C01819=1209.672,408.149,-82.083,-175.808,8.325,148.423
C01820=1209.667,408.397,-82.117,-175.807,8.328,148.423
C01821=1209.664,408.644,-82.152,-175.807,8.330,148.424
C01822=1209.660,408.891,-82.187,-175.807,8.333,148.424
C01823=1209.656,409.139,-82.222,-175.806,8.335,148.425
C01824=1209.651,409.386,-82.257,-175.806,8.337,148.425
C01825=1209.647,409.634,-82.291,-175.806,8.339,148.426
C01826=1209.644,409.882,-82.327,-175.805,8.341,148.426
C01827=1209.639,410.129,-82.361,-175.805,8.343,148.427
C01828=1209.636,410.377,-82.397,-175.804,8.346,148.427
C01829=1209.631,410.624,-82.431,-175.804,8.348,148.428
C01830=1209.627,410.871,-82.467,-175.804,8.350,148.428
C01831=1209.623,411.120,-82.502,-175.803,8.352,148.429
C01832=1209.619,411.366,-82.537,-175.802,8.355,148.429
C01833=1209.615,411.615,-82.572,-175.802,8.357,148.430
C01834=1209.612,411.861,-82.606,-175.802,8.359,148.430
C01835=1209.608,412.109,-82.642,-175.801,8.361,148.430
C01836=1209.604,412.357,-82.677,-175.801,8.364,148.431
C01837=1209.600,412.603,-82.712,-175.801,8.366,148.431
C01838=1209.596,412.852,-82.747,-175.800,8.368,148.432
C01839=1209.592,413.098,-82.782,-175.800,8.370,148.432
C01840=1209.588,413.346,-82.817,-175.800,8.372,148.433
C01841=1209.584,413.594,-82.852,-175.799,8.374,148.433
C01842=1209.579,413.841,-82.887,-175.799,8.377,148.434
C01843=1209.576,414.089,-82.922,-175.798,8.379,148.434
C01844=1209.571,414.336,-82.957,-175.798,8.381,148.435
C01845=1209.567,414.584,-82.992,-175.798,8.383,148.435
C01846=1209.564,414.831,-83.028,-175.797,8.385,148.435
C01847=1209.559,415.079,-83.062,-175.797,8.387,148.436
C01848=1209.556,415.326,-83.098,-175.796,8.390,148.437
C01849=1209.552,415.574,-83.133,-175.796,8.392,148.437
C01850=1209.547,415.821,-83.168,-175.796,8.394,148.437
C01851=1209.544,416.069,-83.204,-175.795,8.396,148.438
C01852=1209.539,416.325,-83.240,-175.795,8.398,148.438
C01853=1209.535,416.581,-83.276,-175.795,8.400,148.439
C01854=1209.533,416.838,-83.312,-175.794,8.402,148.439
C01855=1209.535,417.093,-83.348,-175.794,8.404,148.440
C01856=1209.114,417.093,-83.384,-175.797,8.414,148.443
C01857=1209.112,416.835,-83.348,-175.797,8.413,148.443
C01858=1209.113,416.576,-83.312,-175.798,8.411,148.442
C01859=1209.118,416.317,-83.275,-175.798,8.409,148.442
C01860=1209.122,416.058,-83.238,-175.798,8.407,148.441
C01861=1209.126,415.811,-83.203,-175.799,8.405,148.441
C01862=1209.130,415.563,-83.168,-175.799,8.402,148.441
C01863=1209.134,415.315,-83.133,-175.799,8.400,148.440
C01864=1209.138,415.068,-83.097,-175.800,8.398,148.440
C01865=1209.142,414.820,-83.063,-175.800,8.396,148.439
C01866=1209.146,414.573,-83.027,-175.801,8.394,148.439
C01867=1209.150,414.325,-82.993,-175.801,8.392,148.438
C01868=1209.154,414.078,-82.957,-175.801,8.389,148.438
C01869=1209.158,413.831,-82.922,-175.802,8.387,148.437
C01870=1209.162,413.583,-82.887,-175.802,8.385,148.437
C01871=1209.166,413.335,-82.851,-175.802,8.383,148.436
C01872=1209.170,413.088,-82.817,-175.803,8.381,148.436
C01873=1209.173,412.841,-82.782,-175.803,8.379,148.435
C01874=1209.178,412.593,-82.748,-175.803,8.376,148.435
C01875=1209.181,412.346,-82.712,-175.804,8.374,148.435
C01876=1209.185,412.098,-82.677,-175.804,8.372,148.434
C01877=1209.190,411.851,-82.642,-175.805,8.370,148.434
C01878=1209.193,411.603,-82.607,-175.805,8.368,148.433
C01879=1209.198,411.356,-82.572,-175.805,8.366,148.433
C01880=1209.201,411.108,-82.536,-175.806,8.363,148.432
C01881=1209.205,410.860,-82.502,-175.807,8.360,148.432
C01882=1209.210,410.614,-82.466,-175.807,8.358,148.431
C01883=1209.214,410.365,-82.432,-175.807,8.356,148.431
C01884=1209.218,410.119,-82.396,-175.808,8.354,148.430
C01885=1209.222,409.871,-82.362,-175.808,8.352,148.430
C01886=1209.226,409.623,-82.326,-175.808,8.349,148.429
C01887=1209.230,409.376,-82.292,-175.809,8.347,148.429
C01888=1209.234,409.128,-82.256,-175.809,8.345,148.428
C01889=1209.238,408.881,-82.222,-175.810,8.343,148.428
C01890=1209.242,408.633,-82.186,-175.810,8.341,148.428
C01891=1209.246,408.386,-82.152,-175.810,8.339,148.427
C01892=1209.250,408.138,-82.117,-175.811,8.336,148.426
C01893=1209.253,407.890,-82.082,-175.812,8.334,148.426
C01894=1209.258,407.643,-82.047,-175.812,8.331,148.426
C01895=1209.262,407.396,-82.012,-175.812,8.329,148.425
C01896=1209.266,407.148,-81.977,-175.813,8.327,148.425
C01897=1209.270,406.901,-81.942,-175.813,8.325,148.424
C01898=1209.275,406.653,-81.907,-175.813,8.323,148.424
C01899=1209.278,406.405,-81.872,-175.814,8.320,148.423
C01900=1209.281,406.158,-81.838,-175.814,8.318,148.423
C01901=1209.286,405.910,-81.803,-175.815,8.315,148.422
C01902=1209.290,405.663,-81.768,-175.815,8.313,148.422
C01903=1209.294,405.416,-81.733,-175.816,8.311,148.421
C01904=1209.298,405.167,-81.698,-175.816,8.309,148.421
C01905=1209.302,404.921,-81.663,-175.816,8.306,148.420
C01906=1209.306,404.672,-81.628,-175.817,8.304,148.420
C01907=1209.311,404.426,-81.593,-175.818,8.301,148.419
C01908=1209.314,404.178,-81.559,-175.818,8.299,148.419
C01909=1209.318,403.930,-81.524,-175.819,8.297,148.418
C01910=1209.322,403.683,-81.489,-175.819,8.295,148.418
C01911=1209.326,403.435,-81.454,-175.820,8.292,148.417
C01912=1209.331,403.187,-81.419,-175.820,8.289,148.417
C01913=1209.334,402.940,-81.384,-175.820,8.287,148.416
C01914=1209.338,402.693,-81.350,-175.821,8.285,148.416
C01915=1209.342,402.445,-81.315,-175.821,8.282,148.415
C01916=1209.346,402.198,-81.280,-175.822,8.280,148.415
C01917=1209.350,401.950,-81.245,-175.822,8.278,148.414
C01918=1209.355,401.702,-81.211,-175.822,8.276,148.414
C01919=1209.359,401.455,-81.175,-175.824,8.273,148.414
C01920=1209.362,401.208,-81.141,-175.824,8.271,148.413
C01921=1209.366,400.960,-81.106,-175.824,8.268,148.412
C01922=1209.371,400.712,-81.072,-175.825,8.266,148.412
C01923=1209.375,400.465,-81.036,-175.825,8.263,148.412
C01924=1209.379,400.217,-81.002,-175.826,8.261,148.411
C01925=1209.382,399.969,-80.968,-175.826,8.259,148.411
C01926=1209.387,399.722,-80.933,-175.827,8.256,148.410
C01927=1209.391,399.475,-80.898,-175.827,8.254,148.410
C01928=1209.395,399.227,-80.863,-175.828,8.251,148.409
C01929=1209.399,398.979,-80.828,-175.829,8.248,148.409
C01930=1209.403,398.732,-80.795,-175.829,8.246,148.408
C01931=1209.407,398.484,-80.759,-175.829,8.244,148.408
C01932=1209.411,398.237,-80.725,-175.830,8.241,148.407
C01933=1209.415,397.989,-80.690,-175.831,8.239,148.407
C01934=1209.419,397.742,-80.656,-175.831,8.236,148.406
C01935=1209.423,397.494,-80.620,-175.832,8.234,148.406
C01936=1209.427,397.247,-80.586,-175.832,8.232,148.405
C01937=1209.431,396.999,-80.551,-175.833,8.228,148.405
C01938=1209.435,396.752,-80.517,-175.834,8.226,148.404
C01939=1209.439,396.503,-80.482,-175.834,8.223,148.404
C01940=1209.444,396.256,-80.448,-175.835,8.221,148.403
C01941=1209.447,396.009,-80.412,-175.836,8.218,148.403
C01942=1209.451,395.761,-80.378,-175.836,8.216,148.402
C01943=1209.456,395.514,-80.344,-175.836,8.214,148.402
C01944=1209.460,395.266,-80.309,-175.837,8.211,148.401
C01945=1209.464,395.018,-80.275,-175.838,8.209,148.401
C01946=1209.467,394.771,-80.240,-175.839,8.206,148.400
C01947=1209.472,394.523,-80.206,-175.839,8.204,148.400
C01948=1209.476,394.276,-80.170,-175.840,8.200,148.399
C01949=1209.480,394.029,-80.137,-175.840,8.198,148.399
C01950=1209.484,393.781,-80.102,-175.841,8.195,148.398
C01951=1209.488,393.533,-80.067,-175.841,8.193,148.398
C01952=1209.491,393.285,-80.033,-175.843,8.190,148.397
C01953=1209.497,393.003,-79.994,-175.843,8.187,148.397
C01954=1209.501,392.721,-79.954,-175.844,8.184,148.396
C01955=1209.506,392.439,-79.915,-175.845,8.181,148.395
C01956=1209.510,392.156,-79.876,-175.845,8.179,148.395
C01957=1209.514,391.908,-79.841,-175.846,8.176,148.395
C01958=1209.518,391.661,-79.807,-175.847,8.173,148.394
C01959=1209.523,391.413,-79.773,-175.848,8.171,148.394
C01960=1209.527,391.165,-79.738,-175.848,8.168,148.393
C01961=1209.530,390.918,-79.704,-175.849,8.165,148.392
C01962=1209.534,390.670,-79.669,-175.850,8.163,148.392
C01963=1209.539,390.423,-79.635,-175.851,8.159,148.391
C01964=1209.543,390.176,-79.601,-175.851,8.158,148.391
C01965=1209.547,389.927,-79.566,-175.852,8.154,148.391
C01966=1209.551,389.680,-79.532,-175.853,8.152,148.390
C01967=1209.555,389.432,-79.497,-175.853,8.149,148.390
C01968=1209.559,389.185,-79.463,-175.855,8.147,148.389
C01969=1209.563,388.938,-79.429,-175.855,8.144,148.389
C01970=1209.567,388.690,-79.394,-175.856,8.141,148.388
C01971=1209.572,388.442,-79.360,-175.857,8.138,148.388
C01972=1209.575,388.194,-79.325,-175.857,8.136,148.387
C01973=1209.579,387.947,-79.291,-175.858,8.133,148.387
C01974=1209.583,387.700,-79.257,-175.859,8.130,148.386
C01975=1209.587,387.452,-79.222,-175.860,8.127,148.386
C01976=1209.591,387.205,-79.188,-175.860,8.125,148.385
C01977=1209.595,386.956,-79.154,-175.862,8.122,148.385
C01978=1209.599,386.709,-79.119,-175.862,8.119,148.384
C01979=1209.604,386.461,-79.086,-175.864,8.116,148.384
C01980=1209.608,386.213,-79.051,-175.864,8.114,148.383
C01981=1209.611,385.966,-79.017,-175.865,8.111,148.383
C01982=1209.616,385.719,-78.983,-175.866,8.108,148.382
C01983=1209.619,385.471,-78.949,-175.867,8.105,148.382
C01984=1209.624,385.223,-78.914,-175.868,8.103,148.382
C01985=1209.628,384.976,-78.880,-175.868,8.100,148.381
C01986=1209.632,384.728,-78.846,-175.870,8.097,148.381
C01987=1209.636,384.480,-78.812,-175.870,8.094,148.380
C01988=1209.640,384.233,-78.778,-175.872,8.092,148.380
C01989=1209.644,383.985,-78.744,-175.872,8.089,148.379
C01990=1209.648,383.738,-78.709,-175.873,8.086,148.379
C01991=1209.652,383.491,-78.675,-175.874,8.084,148.378
C01992=1209.656,383.242,-78.641,-175.875,8.081,148.378
C01993=1209.660,382.995,-78.607,-175.876,8.078,148.377
C01994=1209.665,382.747,-78.573,-175.877,8.075,148.377
C01995=1209.668,382.500,-78.538,-175.878,8.072,148.376
C01996=1209.673,382.252,-78.505,-175.879,8.070,148.376
C01997=1209.677,382.004,-78.471,-175.879,8.067,148.375
C01998=1209.681,381.756,-78.436,-175.881,8.064,148.375
C01999=1209.684,381.509,-78.402,-175.882,8.061,148.375
C02000=1209.689,381.261,-78.368,-175.883,8.058,148.374
C02001=1209.692,381.013,-78.334,-175.884,8.055,148.374
C02002=1209.697,380.766,-78.300,-175.885,8.052,148.373
C02003=1209.701,380.518,-78.267,-175.886,8.049,148.373
C02004=1209.705,380.270,-78.232,-175.887,8.046,148.372
C02005=1209.709,380.023,-78.198,-175.888,8.044,148.372
C02006=1209.713,379.775,-78.165,-175.889,8.041,148.371
C02007=1209.718,379.528,-78.130,-175.890,8.038,148.371
C02008=1209.721,379.280,-78.096,-175.891,8.035,148.370
C02009=1209.726,379.032,-78.062,-175.893,8.032,148.370
C02010=1209.730,378.785,-78.028,-175.894,8.029,148.370
C02011=1209.733,378.538,-77.994,-175.894,8.026,148.369
C02012=1209.738,378.289,-77.960,-175.896,8.023,148.369
C02013=1209.742,378.042,-77.926,-175.897,8.021,148.368
C02014=1209.746,377.794,-77.893,-175.898,8.018,148.368
C02015=1209.750,377.546,-77.859,-175.899,8.015,148.368
C02016=1209.753,377.299,-77.825,-175.900,8.012,148.367
C02017=1209.758,377.051,-77.791,-175.901,8.009,148.367
C02018=1209.762,376.804,-77.757,-175.902,8.006,148.366
C02019=1209.766,376.555,-77.723,-175.904,8.003,148.366
C02020=1209.770,376.308,-77.689,-175.905,8.001,148.365
C02021=1209.774,376.060,-77.656,-175.906,7.998,148.365
C02022=1209.778,375.813,-77.622,-175.907,7.995,148.364
C02023=1209.783,375.564,-77.588,-175.908,7.992,148.364
C02024=1209.786,375.317,-77.554,-175.909,7.989,148.364
C02025=1209.790,375.070,-77.520,-175.910,7.986,148.363
C02026=1209.795,374.822,-77.486,-175.912,7.983,148.363
C02027=1209.799,374.574,-77.453,-175.913,7.980,148.362
C02028=1209.802,374.327,-77.419,-175.915,7.977,148.362
C02029=1209.807,374.079,-77.385,-175.916,7.974,148.362
C02030=1209.811,373.831,-77.351,-175.917,7.971,148.361
C02031=1209.815,373.584,-77.318,-175.918,7.968,148.361
C02032=1209.819,373.337,-77.284,-175.919,7.966,148.360
C02033=1209.823,373.088,-77.250,-175.921,7.963,148.360
C02034=1209.827,372.841,-77.216,-175.922,7.959,148.360
C02035=1209.831,372.593,-77.183,-175.924,7.956,148.359
C02036=1209.836,372.345,-77.150,-175.925,7.954,148.359
C02037=1209.840,372.098,-77.116,-175.926,7.951,148.358
C02038=1209.844,371.849,-77.082,-175.927,7.948,148.358
C02039=1209.847,371.602,-77.048,-175.928,7.945,148.358
C02040=1209.852,371.355,-77.015,-175.930,7.942,148.357
C02041=1209.856,371.107,-76.981,-175.931,7.939,148.357
C02042=1209.860,370.859,-76.947,-175.932,7.936,148.356
C02043=1209.864,370.612,-76.914,-175.934,7.933,148.356
C02044=1209.868,370.363,-76.881,-175.935,7.929,148.356
C02045=1209.872,370.116,-76.847,-175.937,7.927,148.355
C02046=1209.877,369.868,-76.813,-175.938,7.924,148.355
C02047=1209.881,369.620,-76.780,-175.939,7.921,148.355
C02048=1209.885,369.373,-76.746,-175.941,7.918,148.354
C02049=1209.889,369.126,-76.713,-175.942,7.915,148.354
C02050=1209.892,368.877,-76.679,-175.944,7.912,148.353
C02051=1209.896,368.629,-76.646,-175.945,7.909,148.353
C02052=1209.901,368.382,-76.612,-175.947,7.906,148.353
C02053=1209.905,368.134,-76.579,-175.948,7.903,148.352
C02054=1209.909,367.887,-76.545,-175.949,7.900,148.352
C02055=1209.913,367.639,-76.512,-175.951,7.897,148.352
C02056=1209.918,367.391,-76.479,-175.952,7.894,148.351
C02057=1209.922,367.110,-76.441,-175.954,7.891,148.351
C02058=1209.927,366.831,-76.403,-175.955,7.887,148.350
C02059=1209.931,366.551,-76.365,-175.958,7.884,148.350
C02060=1209.936,366.269,-76.327,-175.959,7.880,148.350
C02061=1209.940,366.022,-76.294,-175.961,7.877,148.349
C02062=1209.944,365.775,-76.260,-175.962,7.875,148.349
C02063=1209.948,365.527,-76.227,-175.964,7.871,148.349
C02064=1209.952,365.279,-76.194,-175.965,7.869,148.348
C02065=1209.956,365.031,-76.161,-175.966,7.866,148.348
C02066=1209.960,364.784,-76.128,-175.969,7.862,148.348
C02067=1209.965,364.536,-76.095,-175.970,7.860,148.347
C02068=1209.969,364.288,-76.061,-175.971,7.857,148.347
C02069=1209.973,364.040,-76.028,-175.973,7.853,148.347
C02070=1209.977,363.793,-75.995,-175.974,7.851,148.346
C02071=1209.980,363.545,-75.961,-175.976,7.847,148.346
C02072=1209.984,363.297,-75.928,-175.978,7.844,148.346
C02073=1209.989,363.049,-75.895,-175.979,7.842,148.345
C02074=1209.993,362.802,-75.861,-175.981,7.838,148.345
C02075=1209.997,362.554,-75.828,-175.982,7.835,148.345
C02076=1210.001,362.306,-75.795,-175.985,7.832,148.344
C02077=1210.005,362.059,-75.762,-175.986,7.829,148.344
C02078=1210.009,361.811,-75.729,-175.987,7.826,148.344
C02079=1210.013,361.563,-75.696,-175.989,7.823,148.343
C02080=1210.018,361.315,-75.663,-175.990,7.820,148.343
C02081=1210.022,361.067,-75.630,-175.993,7.817,148.343
C02082=1210.026,360.819,-75.597,-175.994,7.814,148.342
C02083=1210.030,360.572,-75.564,-175.995,7.812,148.342
C02084=1210.034,360.324,-75.531,-175.997,7.808,148.342
C02085=1210.039,360.076,-75.497,-175.999,7.805,148.341
C02086=1210.043,359.828,-75.464,-176.001,7.802,148.341
C02087=1210.047,359.581,-75.431,-176.002,7.799,148.341
C02088=1210.051,359.333,-75.398,-176.004,7.796,148.341
C02089=1210.055,359.085,-75.365,-176.006,7.793,148.340
C02090=1210.059,358.837,-75.332,-176.007,7.791,148.340
C02091=1210.063,358.589,-75.300,-176.009,7.787,148.340
C02092=1210.067,358.342,-75.267,-176.011,7.784,148.339
C02093=1210.071,358.094,-75.234,-176.013,7.781,148.339
C02094=1210.075,357.846,-75.200,-176.014,7.778,148.339
C02095=1210.079,357.598,-75.167,-176.016,7.775,148.339
C02096=1210.084,357.350,-75.135,-176.018,7.772,148.338
C02097=1210.088,357.102,-75.102,-176.020,7.769,148.338
C02098=1210.091,356.855,-75.069,-176.021,7.766,148.338
C02099=1210.096,356.607,-75.036,-176.023,7.763,148.337
C02100=1210.100,356.359,-75.003,-176.025,7.760,148.337
C02101=1210.104,356.111,-74.970,-176.027,7.757,148.337
C02102=1210.108,355.863,-74.937,-176.029,7.754,148.337
C02103=1210.113,355.616,-74.904,-176.030,7.751,148.336
C02104=1210.117,355.368,-74.873,-176.032,7.748,148.336
C02105=1210.121,355.121,-74.839,-176.034,7.745,148.336
C02106=1210.125,354.873,-74.806,-176.035,7.742,148.335
C02107=1210.129,354.625,-74.774,-176.038,7.739,148.335
C02108=1210.134,354.377,-74.741,-176.039,7.736,148.335
C02109=1210.137,354.129,-74.708,-176.041,7.734,148.335
C02110=1210.141,353.881,-74.676,-176.043,7.730,148.334
C02111=1210.146,353.633,-74.642,-176.044,7.727,148.334
C02112=1210.150,353.385,-74.610,-176.047,7.724,148.334
C02113=1210.153,353.138,-74.577,-176.048,7.722,148.334
C02114=1210.158,352.891,-74.545,-176.050,7.718,148.334
C02115=1210.163,352.642,-74.512,-176.052,7.715,148.333
C02116=1210.167,352.394,-74.479,-176.054,7.712,148.333
C02117=1210.170,352.146,-74.447,-176.055,7.710,148.333
C02118=1210.175,351.899,-74.414,-176.058,7.706,148.333
C02119=1210.179,351.650,-74.382,-176.059,7.704,148.332
C02120=1210.182,351.403,-74.349,-176.061,7.700,148.332
C02121=1210.187,351.155,-74.317,-176.063,7.697,148.332
C02122=1210.192,350.908,-74.284,-176.065,7.694,148.332
C02123=1210.195,350.660,-74.252,-176.067,7.692,148.331
C02124=1210.199,350.412,-74.219,-176.069,7.688,148.331
C02125=1210.204,350.163,-74.186,-176.070,7.686,148.331
C02126=1210.207,349.916,-74.154,-176.073,7.682,148.331
C02127=1210.212,349.668,-74.121,-176.075,7.679,148.331
C02128=1210.216,349.421,-74.089,-176.076,7.677,148.330
C02129=1210.220,349.173,-74.057,-176.079,7.673,148.330
C02130=1210.225,348.924,-74.024,-176.080,7.671,148.330
C02131=1210.229,348.677,-73.991,-176.082,7.667,148.330
C02132=1210.232,348.428,-73.959,-176.084,7.665,148.329
C02133=1210.237,348.181,-73.927,-176.086,7.661,148.329
C02134=1210.241,347.933,-73.895,-176.088,7.659,148.329
C02135=1210.245,347.685,-73.862,-176.090,7.655,148.329
C02136=1210.250,347.437,-73.829,-176.091,7.653,148.329
C02137=1210.253,347.189,-73.797,-176.094,7.649,148.328
C02138=1210.258,346.942,-73.765,-176.095,7.647,148.328
C02139=1210.262,346.694,-73.733,-176.098,7.644,148.328
C02140=1210.266,346.446,-73.700,-176.099,7.641,148.328
C02141=1210.270,346.198,-73.668,-176.101,7.638,148.328
C02142=1210.275,345.950,-73.636,-176.103,7.635,148.327
C02143=1210.279,345.702,-73.603,-176.105,7.632,148.327
C02144=1210.283,345.454,-73.571,-176.107,7.629,148.327
C02145=1210.287,345.206,-73.539,-176.109,7.626,148.327
C02146=1210.291,344.959,-73.507,-176.111,7.624,148.327
C02147=1210.296,344.711,-73.474,-176.113,7.620,148.327
C02148=1210.299,344.463,-73.442,-176.116,7.617,148.326
C02149=1210.304,344.215,-73.410,-176.117,7.615,148.326
C02150=1210.308,343.967,-73.378,-176.119,7.611,148.326
C02151=1210.313,343.719,-73.346,-176.121,7.609,148.326
C02152=1210.316,343.472,-73.313,-176.123,7.605,148.325
C02153=1210.320,343.223,-73.281,-176.125,7.603,148.325
C02154=1210.325,342.976,-73.249,-176.127,7.600,148.325
C02155=1210.328,342.728,-73.218,-176.129,7.597,148.325
C02156=1210.333,342.479,-73.185,-176.131,7.594,148.325
C02157=1210.337,342.232,-73.154,-176.133,7.591,148.325
C02158=1210.342,341.984,-73.121,-176.135,7.588,148.324
C02159=1210.345,341.736,-73.089,-176.138,7.585,148.324
C02160=1210.350,341.488,-73.057,-176.139,7.582,148.324
C02161=1210.354,341.210,-73.021,-176.141,7.579,148.324
C02162=1210.359,340.932,-72.985,-176.144,7.576,148.324
C02163=1210.364,340.654,-72.949,-176.146,7.572,148.324
C02164=1210.368,340.375,-72.914,-176.149,7.569,148.323
C02165=1210.372,340.128,-72.882,-176.151,7.566,148.323
C02166=1210.377,339.880,-72.850,-176.152,7.563,148.323
C02167=1210.381,339.632,-72.818,-176.155,7.560,148.323
C02168=1210.386,339.384,-72.786,-176.157,7.558,148.323
C02169=1210.389,339.136,-72.754,-176.159,7.554,148.323
C02170=1210.393,338.888,-72.722,-176.161,7.552,148.322
C02171=1210.398,338.640,-72.690,-176.163,7.549,148.322
C02172=1210.402,338.392,-72.658,-176.165,7.546,148.322
C02173=1210.406,338.145,-72.627,-176.167,7.543,148.322
C02174=1210.410,337.897,-72.595,-176.169,7.540,148.322
C02175=1210.414,337.648,-72.563,-176.171,7.537,148.322
C02176=1210.419,337.401,-72.531,-176.174,7.534,148.322
C02177=1210.423,337.152,-72.500,-176.175,7.532,148.321
C02178=1210.427,336.904,-72.467,-176.177,7.528,148.321
C02179=1210.431,336.657,-72.436,-176.180,7.526,148.321
C02180=1210.435,336.409,-72.404,-176.182,7.523,148.321
C02181=1210.439,336.161,-72.373,-176.183,7.520,148.321
C02182=1210.444,335.913,-72.340,-176.186,7.517,148.321
C02183=1210.448,335.664,-72.309,-176.188,7.514,148.321
C02184=1210.452,335.417,-72.278,-176.190,7.511,148.320
C02185=1210.456,335.169,-72.246,-176.193,7.508,148.320
C02186=1210.460,334.922,-72.214,-176.194,7.506,148.320
C02187=1210.465,334.673,-72.183,-176.197,7.502,148.320
C02188=1210.469,334.425,-72.151,-176.199,7.500,148.320
C02189=1210.473,334.177,-72.119,-176.201,7.497,148.320
C02190=1210.477,333.929,-72.087,-176.202,7.494,148.320
C02191=1210.481,333.681,-72.057,-176.205,7.491,148.320
C02192=1210.486,333.433,-72.024,-176.207,7.488,148.319
C02193=1210.490,333.186,-71.993,-176.209,7.485,148.319
C02194=1210.494,332.937,-71.962,-176.212,7.482,148.319
C02195=1210.498,332.690,-71.930,-176.213,7.480,148.319
C02196=1210.502,332.442,-71.898,-176.216,7.477,148.319
C02197=1210.507,332.194,-71.867,-176.218,7.474,148.319
C02198=1210.510,331.946,-71.836,-176.220,7.471,148.319
C02199=1210.516,331.697,-71.804,-176.223,7.468,148.319
C02200=1210.519,331.449,-71.772,-176.224,7.465,148.319
C02201=1210.524,331.202,-71.741,-176.227,7.462,148.319
C02202=1210.528,330.953,-71.710,-176.229,7.460,148.318
C02203=1210.532,330.706,-71.678,-176.231,7.457,148.318
C02204=1210.536,330.457,-71.647,-176.233,7.454,148.318
C02205=1210.540,330.210,-71.616,-176.236,7.451,148.318
C02206=1210.544,329.961,-71.585,-176.237,7.449,148.318
C02207=1210.549,329.714,-71.553,-176.240,7.446,148.318
C02208=1210.553,329.465,-71.522,-176.242,7.442,148.318
C02209=1210.557,329.218,-71.491,-176.244,7.440,148.318
C02210=1210.561,328.969,-71.459,-176.246,7.437,148.318
C02211=1210.565,328.722,-71.428,-176.248,7.434,148.317
C02212=1210.569,328.473,-71.397,-176.251,7.431,148.317
C02213=1210.574,328.226,-71.365,-176.253,7.429,148.317
C02214=1210.578,327.977,-71.334,-176.255,7.426,148.317
C02215=1210.582,327.730,-71.303,-176.258,7.423,148.317
C02216=1210.587,327.482,-71.272,-176.259,7.420,148.317
C02217=1210.591,327.233,-71.241,-176.262,7.417,148.317
C02218=1210.595,326.986,-71.209,-176.264,7.415,148.317
C02219=1210.599,326.737,-71.178,-176.266,7.411,148.317
C02220=1210.603,326.489,-71.147,-176.268,7.409,148.317
C02221=1210.607,326.241,-71.116,-176.271,7.406,148.317
C02222=1210.612,325.993,-71.085,-176.273,7.403,148.317
C02223=1210.616,325.745,-71.054,-176.275,7.400,148.317
C02224=1210.620,325.497,-71.022,-176.278,7.397,148.317
C02225=1210.625,325.249,-70.991,-176.279,7.395,148.316
C02226=1210.629,325.001,-70.960,-176.282,7.392,148.316
C02227=1210.633,324.753,-70.929,-176.284,7.389,148.316
C02228=1210.637,324.506,-70.899,-176.286,7.386,148.316
C02229=1210.641,324.257,-70.868,-176.288,7.384,148.316
C02230=1210.646,324.009,-70.837,-176.291,7.381,148.316
C02231=1210.649,323.761,-70.805,-176.293,7.378,148.316
C02232=1210.654,323.513,-70.774,-176.295,7.375,148.316
C02233=1210.659,323.265,-70.743,-176.298,7.372,148.316
C02234=1210.663,323.017,-70.712,-176.300,7.370,148.316
C02235=1210.666,322.769,-70.682,-176.302,7.367,148.316
C02236=1210.671,322.522,-70.651,-176.304,7.364,148.316
C02237=1210.675,322.273,-70.620,-176.306,7.361,148.316
C02238=1210.679,322.025,-70.589,-176.309,7.358,148.316
C02239=1210.684,321.777,-70.558,-176.311,7.356,148.316
C02240=1210.688,321.528,-70.527,-176.313,7.352,148.315
C02241=1210.692,321.281,-70.497,-176.315,7.350,148.315
C02242=1210.696,321.033,-70.466,-176.318,7.347,148.315
C02243=1210.700,320.784,-70.435,-176.320,7.345,148.315
C02244=1210.705,320.537,-70.403,-176.322,7.342,148.315
C02245=1210.709,320.289,-70.373,-176.325,7.339,148.315
C02246=1210.713,320.040,-70.342,-176.327,7.336,148.315
C02247=1210.717,319.792,-70.311,-176.329,7.333,148.315
C02248=1210.722,319.545,-70.280,-176.332,7.331,148.315
C02249=1210.725,319.296,-70.250,-176.334,7.328,148.315
C02250=1210.730,319.048,-70.219,-176.336,7.325,148.315
C02251=1210.734,318.800,-70.188,-176.339,7.322,148.315
C02252=1210.739,318.552,-70.158,-176.341,7.320,148.315
C02253=1210.742,318.304,-70.127,-176.343,7.317,148.315
C02254=1210.747,318.056,-70.096,-176.346,7.314,148.315
C02255=1210.751,317.808,-70.066,-176.348,7.311,148.315
C02256=1210.755,317.560,-70.035,-176.350,7.308,148.315
C02257=1210.760,317.311,-70.005,-176.352,7.306,148.315
C02258=1210.764,317.063,-69.974,-176.355,7.303,148.315
C02259=1210.768,316.815,-69.944,-176.357,7.301,148.315
C02260=1210.773,316.568,-69.913,-176.359,7.298,148.315
C02261=1210.777,316.319,-69.882,-176.362,7.295,148.315
C02262=1210.781,316.071,-69.852,-176.364,7.292,148.315
C02263=1210.785,315.823,-69.821,-176.366,7.289,148.315
C02264=1210.789,315.576,-69.791,-176.369,7.287,148.315
C02265=1210.794,315.299,-69.758,-176.371,7.284,148.315
C02266=1210.798,315.023,-69.723,-176.374,7.281,148.315
C02267=1210.804,314.746,-69.689,-176.377,7.278,148.315
C02268=1210.808,314.471,-69.655,-176.379,7.274,148.314
C02269=1210.812,314.223,-69.625,-176.381,7.272,148.314
C02270=1210.817,313.974,-69.595,-176.384,7.269,148.314
C02271=1210.821,313.727,-69.565,-176.386,7.266,148.314
C02272=1210.826,313.479,-69.534,-176.388,7.264,148.315
C02273=1210.830,313.230,-69.503,-176.391,7.260,148.314
C02274=1210.834,312.982,-69.473,-176.393,7.258,148.314
C02275=1210.838,312.734,-69.443,-176.395,7.255,148.314
C02276=1210.842,312.486,-69.412,-176.398,7.253,148.314
C02277=1210.847,312.238,-69.382,-176.400,7.250,148.314
C02278=1210.851,311.990,-69.352,-176.402,7.248,148.315
C02279=1210.855,311.741,-69.321,-176.405,7.245,148.315
C02280=1210.859,311.493,-69.292,-176.407,7.242,148.314
C02281=1210.864,311.245,-69.261,-176.409,7.239,148.314
C02282=1210.868,310.997,-69.231,-176.411,7.237,148.314
C02283=1210.873,310.749,-69.201,-176.414,7.234,148.314
C02284=1210.877,310.501,-69.170,-176.417,7.231,148.314
C02285=1210.881,310.253,-69.141,-176.419,7.229,148.314
C02286=1210.885,310.005,-69.110,-176.422,7.226,148.314
C02287=1210.889,309.756,-69.080,-176.424,7.223,148.315
C02288=1210.894,309.508,-69.050,-176.426,7.220,148.314
C02289=1210.898,309.260,-69.020,-176.428,7.218,148.314
C02290=1210.902,309.012,-68.989,-176.431,7.215,148.314
C02291=1210.906,308.764,-68.960,-176.433,7.213,148.314
C02292=1210.910,308.516,-68.930,-176.436,7.210,148.314
C02293=1210.915,308.267,-68.900,-176.438,7.207,148.315
C02294=1210.919,308.020,-68.870,-176.440,7.204,148.315
C02295=1210.924,307.771,-68.840,-176.442,7.202,148.315
C02296=1210.928,307.523,-68.809,-176.445,7.199,148.315
C02297=1210.932,307.275,-68.780,-176.447,7.197,148.315
C02298=1210.937,307.027,-68.749,-176.450,7.194,148.315
C02299=1210.941,306.779,-68.720,-176.453,7.191,148.315
C02300=1210.945,306.530,-68.690,-176.455,7.189,148.315
C02301=1210.949,306.282,-68.659,-176.457,7.186,148.315
C02302=1210.953,306.034,-68.630,-176.459,7.183,148.315
C02303=1210.957,305.785,-68.600,-176.462,7.180,148.315
C02304=1210.962,305.538,-68.569,-176.464,7.178,148.315
C02305=1210.966,305.289,-68.540,-176.467,7.175,148.315
C02306=1210.970,305.041,-68.511,-176.469,7.173,148.315
C02307=1210.975,304.793,-68.480,-176.471,7.170,148.315
C02308=1210.979,304.545,-68.450,-176.473,7.167,148.315
C02309=1210.983,304.296,-68.421,-176.476,7.164,148.315
C02310=1210.987,304.049,-68.391,-176.478,7.162,148.315
C02311=1210.992,303.800,-68.361,-176.481,7.159,148.315
C02312=1210.996,303.552,-68.331,-176.483,7.157,148.315
C02313=1211.001,303.304,-68.302,-176.486,7.154,148.315
C02314=1211.004,303.056,-68.272,-176.488,7.152,148.315
C02315=1211.009,302.807,-68.241,-176.491,7.149,148.315
C02316=1211.014,302.559,-68.212,-176.493,7.147,148.315
C02317=1211.018,302.311,-68.183,-176.495,7.143,148.315
C02318=1211.022,302.063,-68.153,-176.497,7.141,148.315
C02319=1211.026,301.815,-68.123,-176.500,7.138,148.315
C02320=1211.031,301.567,-68.093,-176.502,7.136,148.315
C02321=1211.036,301.319,-68.064,-176.505,7.133,148.315
C02322=1211.040,301.071,-68.034,-176.507,7.131,148.315
C02323=1211.044,300.822,-68.005,-176.510,7.128,148.315
C02324=1211.048,300.574,-67.975,-176.512,7.126,148.316
C02325=1211.052,300.326,-67.946,-176.515,7.123,148.316
C02326=1211.057,300.077,-67.916,-176.517,7.121,148.316
C02327=1211.061,299.829,-67.887,-176.520,7.118,148.316
C02328=1211.066,299.581,-67.857,-176.522,7.115,148.316
C02329=1211.070,299.332,-67.828,-176.525,7.112,148.316
C02330=1211.074,299.085,-67.797,-176.527,7.110,148.316
C02331=1211.078,298.837,-67.768,-176.529,7.107,148.316
C02332=1211.082,298.588,-67.739,-176.532,7.105,148.316
C02333=1211.087,298.341,-67.709,-176.534,7.102,148.316
C02334=1211.091,298.092,-67.680,-176.536,7.100,148.316
C02335=1211.095,297.844,-67.651,-176.539,7.097,148.316
C02336=1211.100,297.595,-67.622,-176.541,7.094,148.316
C02337=1211.104,297.347,-67.592,-176.544,7.091,148.316
C02338=1211.109,297.098,-67.562,-176.546,7.090,148.316
C02339=1211.113,296.850,-67.533,-176.549,7.087,148.316
C02340=1211.117,296.602,-67.503,-176.551,7.084,148.316
C02341=1211.121,296.354,-67.474,-176.554,7.081,148.316
C02342=1211.126,296.106,-67.445,-176.556,7.079,148.316
C02343=1211.130,295.858,-67.415,-176.559,7.076,148.316
C02344=1211.134,295.610,-67.386,-176.561,7.074,148.317
C02345=1211.139,295.361,-67.356,-176.564,7.071,148.317
C02346=1211.143,295.112,-67.328,-176.566,7.069,148.317
C02347=1211.147,294.864,-67.298,-176.569,7.066,148.317
C02348=1211.151,294.617,-67.270,-176.571,7.064,148.317
C02349=1211.155,294.369,-67.240,-176.574,7.061,148.317
C02350=1211.160,294.120,-67.211,-176.576,7.058,148.317
C02351=1211.164,293.871,-67.182,-176.578,7.055,148.317
C02352=1211.168,293.623,-67.153,-176.581,7.053,148.317
C02353=1211.172,293.375,-67.123,-176.583,7.051,148.317
C02354=1211.177,293.127,-67.094,-176.586,7.048,148.317
C02355=1211.182,292.878,-67.065,-176.588,7.046,148.317
C02356=1211.186,292.630,-67.036,-176.591,7.043,148.317
C02357=1211.190,292.382,-67.007,-176.593,7.041,148.318
C02358=1211.194,292.134,-66.977,-176.595,7.038,148.318
C02359=1211.199,291.885,-66.949,-176.598,7.036,148.318
C02360=1211.203,291.638,-66.920,-176.601,7.033,148.318
C02361=1211.207,291.389,-66.890,-176.603,7.031,148.318
C02362=1211.211,291.140,-66.862,-176.606,7.028,148.318
C02363=1211.216,290.893,-66.833,-176.608,7.026,148.318
C02364=1211.220,290.645,-66.803,-176.610,7.023,148.318
C02365=1211.225,290.396,-66.774,-176.613,7.021,148.318
C02366=1211.228,290.148,-66.746,-176.615,7.018,148.318
C02367=1211.233,289.899,-66.717,-176.618,7.015,148.318
C02368=1211.238,289.651,-66.688,-176.620,7.013,148.318
C02369=1211.242,289.377,-66.656,-176.623,7.010,148.318
C02370=1211.247,289.102,-66.624,-176.626,7.007,148.319
C02371=1211.252,288.829,-66.592,-176.628,7.004,148.319
C02372=1211.257,288.554,-66.560,-176.631,7.001,148.319
C02373=1211.261,288.306,-66.531,-176.634,7.000,148.319
C02374=1211.265,288.057,-66.502,-176.636,6.997,148.319
C02375=1211.270,287.810,-66.473,-176.639,6.994,148.319
C02376=1211.275,287.561,-66.444,-176.641,6.992,148.319
C02377=1211.278,287.312,-66.416,-176.644,6.989,148.319
C02378=1211.283,287.065,-66.387,-176.646,6.987,148.320
C02379=1211.288,286.816,-66.358,-176.649,6.984,148.320
C02380=1211.291,286.568,-66.330,-176.651,6.982,148.320
C02381=1211.296,286.320,-66.301,-176.653,6.980,148.320
C02382=1211.300,286.071,-66.272,-176.656,6.977,148.320
C02383=1211.305,285.822,-66.243,-176.658,6.975,148.320
C02384=1211.309,285.575,-66.215,-176.661,6.972,148.320
C02385=1211.313,285.326,-66.186,-176.663,6.970,148.320
C02386=1211.318,285.077,-66.157,-176.666,6.967,148.320
C02387=1211.322,284.830,-66.129,-176.668,6.965,148.320
C02388=1211.326,284.581,-66.100,-176.670,6.963,148.320
C02389=1211.331,284.332,-66.071,-176.674,6.960,148.321
C02390=1211.335,284.085,-66.043,-176.676,6.958,148.321
C02391=1211.339,283.836,-66.014,-176.678,6.955,148.321
C02392=1211.344,283.588,-65.986,-176.681,6.952,148.321
C02393=1211.348,283.339,-65.957,-176.684,6.950,148.321
C02394=1211.352,283.091,-65.928,-176.686,6.947,148.321
C02395=1211.357,282.843,-65.900,-176.688,6.945,148.321
C02396=1211.361,282.594,-65.871,-176.691,6.943,148.321
C02397=1211.366,282.347,-65.844,-176.693,6.940,148.322
C02398=1211.370,282.098,-65.815,-176.696,6.937,148.322
C02399=1211.374,281.849,-65.785,-176.698,6.935,148.322
C02400=1211.379,281.602,-65.758,-176.701,6.933,148.322
C02401=1211.383,281.353,-65.729,-176.703,6.930,148.322
C02402=1211.387,281.105,-65.701,-176.705,6.928,148.322
C02403=1211.392,280.856,-65.672,-176.709,6.925,148.322
C02404=1211.396,280.608,-65.645,-176.711,6.923,148.322
C02405=1211.400,280.360,-65.615,-176.713,6.921,148.322
C02406=1211.404,280.111,-65.587,-176.716,6.918,148.323
C02407=1211.409,279.863,-65.559,-176.718,6.916,148.323
C02408=1211.413,279.614,-65.530,-176.721,6.913,148.323
C02409=1211.418,279.366,-65.502,-176.723,6.911,148.323
C02410=1211.422,279.118,-65.474,-176.726,6.909,148.323
C02411=1211.427,278.869,-65.446,-176.728,6.906,148.323
C02412=1211.431,278.621,-65.417,-176.731,6.904,148.323
C02413=1211.436,278.373,-65.389,-176.733,6.902,148.324
C02414=1211.439,278.124,-65.361,-176.736,6.899,148.324
C02415=1211.444,277.876,-65.333,-176.738,6.897,148.324
C02416=1211.448,277.627,-65.304,-176.741,6.894,148.324
C02417=1211.453,277.380,-65.277,-176.743,6.892,148.324
C02418=1211.457,277.131,-65.248,-176.746,6.890,148.324
C02419=1211.462,276.883,-65.220,-176.748,6.887,148.324
C02420=1211.466,276.634,-65.191,-176.751,6.885,148.324
C02421=1211.470,276.386,-65.164,-176.753,6.883,148.325
C02422=1211.474,276.137,-65.135,-176.756,6.880,148.325
C02423=1211.479,275.889,-65.107,-176.758,6.878,148.325
C02424=1211.483,275.641,-65.079,-176.761,6.875,148.325
C02425=1211.487,275.393,-65.051,-176.763,6.873,148.325
C02426=1211.492,275.144,-65.022,-176.766,6.871,148.325
C02427=1211.496,274.895,-64.995,-176.769,6.868,148.325
C02428=1211.500,274.647,-64.967,-176.771,6.866,148.325
C02429=1211.505,274.399,-64.939,-176.773,6.864,148.326
C02430=1211.509,274.150,-64.911,-176.776,6.861,148.326
C02431=1211.513,273.902,-64.883,-176.778,6.858,148.326
C02432=1211.518,273.654,-64.855,-176.781,6.857,148.326
C02433=1211.523,273.405,-64.827,-176.783,6.854,148.326
C02434=1211.527,273.157,-64.799,-176.786,6.852,148.327
C02435=1211.531,272.908,-64.771,-176.788,6.850,148.327
C02436=1211.536,272.660,-64.743,-176.791,6.846,148.327
C02437=1211.540,272.412,-64.715,-176.794,6.845,148.327
C02438=1211.544,272.163,-64.688,-176.796,6.842,148.327
C02439=1211.549,271.915,-64.659,-176.799,6.840,148.327
C02440=1211.553,271.666,-64.631,-176.801,6.838,148.327
C02441=1211.558,271.418,-64.604,-176.803,6.835,148.327
C02442=1211.562,271.170,-64.576,-176.806,6.833,148.328
C02443=1211.566,270.921,-64.548,-176.808,6.830,148.328
C02444=1211.571,270.673,-64.520,-176.811,6.829,148.328
C02445=1211.575,270.424,-64.492,-176.814,6.826,148.328
C02446=1211.579,270.176,-64.465,-176.816,6.824,148.328
C02447=1211.584,269.928,-64.438,-176.818,6.821,148.328
C02448=1211.588,269.679,-64.409,-176.821,6.818,148.328
C02449=1211.593,269.431,-64.381,-176.824,6.817,148.329
C02450=1211.597,269.182,-64.354,-176.826,6.814,148.329
C02451=1211.601,268.934,-64.326,-176.829,6.812,148.329
C02452=1211.606,268.685,-64.299,-176.831,6.809,148.329
C02453=1211.610,268.437,-64.271,-176.834,6.808,148.329
C02454=1211.615,268.188,-64.243,-176.836,6.805,148.330
C02455=1211.619,267.940,-64.215,-176.839,6.803,148.330
C02456=1211.624,267.692,-64.187,-176.841,6.801,148.330
C02457=1211.628,267.443,-64.160,-176.844,6.798,148.330
C02458=1211.632,267.195,-64.132,-176.847,6.796,148.330
C02459=1211.637,266.947,-64.105,-176.849,6.793,148.330
C02460=1211.640,266.698,-64.077,-176.852,6.791,148.331
C02461=1211.645,266.449,-64.050,-176.854,6.789,148.331
C02462=1211.650,266.201,-64.023,-176.857,6.787,148.331
C02463=1211.655,265.953,-63.994,-176.859,6.784,148.331
C02464=1211.659,265.704,-63.967,-176.862,6.782,148.331
C02465=1211.663,265.456,-63.939,-176.864,6.780,148.331
C02466=1211.668,265.207,-63.912,-176.867,6.778,148.332
C02467=1211.672,264.959,-63.884,-176.869,6.775,148.332
C02468=1211.676,264.710,-63.857,-176.872,6.773,148.332
C02469=1211.681,264.462,-63.830,-176.874,6.771,148.332
C02470=1211.685,264.214,-63.802,-176.877,6.769,148.332
C02471=1211.689,263.965,-63.775,-176.879,6.766,148.332
C02472=1211.694,263.716,-63.748,-176.882,6.764,148.333
C02473=1211.699,263.444,-63.718,-176.885,6.761,148.333
C02474=1211.704,263.171,-63.688,-176.887,6.759,148.333
C02475=1211.708,262.899,-63.658,-176.890,6.756,148.333
C02476=1211.713,262.626,-63.627,-176.893,6.754,148.333
C02477=1211.718,262.377,-63.600,-176.896,6.751,148.334
C02478=1211.722,262.129,-63.573,-176.898,6.749,148.334
C02479=1211.727,261.881,-63.545,-176.901,6.747,148.334
C02480=1211.731,261.632,-63.518,-176.903,6.744,148.334
C02481=1211.735,261.383,-63.491,-176.906,6.742,148.334
C02482=1211.740,261.134,-63.464,-176.908,6.740,148.334
C02483=1211.744,260.887,-63.436,-176.911,6.738,148.335
C02484=1211.748,260.638,-63.410,-176.913,6.735,148.335
C02485=1211.753,260.390,-63.382,-176.916,6.734,148.335
C02486=1211.757,260.141,-63.355,-176.918,6.731,148.335
C02487=1211.762,259.892,-63.328,-176.921,6.729,148.336
C02488=1211.766,259.644,-63.301,-176.923,6.726,148.336
C02489=1211.771,259.396,-63.273,-176.926,6.725,148.336
C02490=1211.775,259.147,-63.246,-176.928,6.722,148.336
C02491=1211.780,258.899,-63.219,-176.931,6.721,148.336
C02492=1211.783,258.650,-63.192,-176.933,6.717,148.336
C02493=1211.788,258.401,-63.165,-176.936,6.716,148.337
C02494=1211.793,258.153,-63.138,-176.939,6.714,148.337
C02495=1211.797,257.905,-63.111,-176.941,6.712,148.337
C02496=1211.802,257.656,-63.084,-176.944,6.709,148.337
C02497=1211.807,257.408,-63.057,-176.946,6.707,148.337
C02498=1211.811,257.159,-63.030,-176.949,6.705,148.338
C02499=1211.815,256.910,-63.003,-176.951,6.703,148.338
C02500=1211.819,256.662,-62.976,-176.954,6.700,148.338
C02501=1211.824,256.413,-62.949,-176.956,6.698,148.338
C02502=1211.828,256.165,-62.922,-176.959,6.696,148.338
C02503=1211.832,255.916,-62.895,-176.961,6.694,148.339
C02504=1211.837,255.668,-62.868,-176.964,6.691,148.339
C02505=1211.842,255.419,-62.841,-176.967,6.689,148.339
C02506=1211.846,255.171,-62.815,-176.969,6.687,148.339
C02507=1211.850,254.923,-62.788,-176.971,6.685,148.339
C02508=1211.855,254.674,-62.761,-176.974,6.683,148.340
C02509=1211.860,254.426,-62.734,-176.977,6.680,148.340
C02510=1211.863,254.177,-62.707,-176.979,6.678,148.340
C02511=1211.868,253.928,-62.680,-176.982,6.676,148.340
C02512=1211.872,253.680,-62.653,-176.984,6.674,148.341
C02513=1211.877,253.431,-62.627,-176.987,6.671,148.341
C02514=1211.881,253.183,-62.600,-176.989,6.669,148.341
C02515=1211.886,252.934,-62.573,-176.992,6.667,148.341
C02516=1211.890,252.686,-62.546,-176.994,6.665,148.341
C02517=1211.894,252.437,-62.519,-176.997,6.664,148.342
C02518=1211.899,252.189,-62.492,-177.000,6.660,148.342
C02519=1211.903,251.940,-62.466,-177.002,6.659,148.342
C02520=1211.908,251.692,-62.439,-177.004,6.656,148.342
C02521=1211.913,251.443,-62.412,-177.007,6.655,148.342
C02522=1211.917,251.195,-62.386,-177.010,6.653,148.343
C02523=1211.921,250.946,-62.359,-177.012,6.650,148.343
C02524=1211.925,250.698,-62.333,-177.015,6.648,148.343
C02525=1211.930,250.449,-62.306,-177.017,6.646,148.343
C02526=1211.935,250.201,-62.279,-177.020,6.644,148.343
C02527=1211.939,249.952,-62.253,-177.022,6.642,148.344
C02528=1211.944,249.703,-62.226,-177.025,6.639,148.344
C02529=1211.948,249.455,-62.200,-177.028,6.637,148.344
C02530=1211.952,249.206,-62.173,-177.030,6.635,148.344
C02531=1211.956,248.958,-62.147,-177.032,6.633,148.344
C02532=1211.961,248.709,-62.120,-177.035,6.631,148.345
C02533=1211.966,248.460,-62.093,-177.038,6.628,148.345
C02534=1211.970,248.212,-62.067,-177.040,6.626,148.345
C02535=1211.975,247.963,-62.041,-177.043,6.624,148.345
C02536=1211.979,247.715,-62.014,-177.045,6.622,148.346
C02537=1211.983,247.466,-61.987,-177.048,6.620,148.346
C02538=1211.988,247.217,-61.961,-177.050,6.619,148.346
C02539=1211.993,246.970,-61.935,-177.053,6.615,148.346
C02540=1211.997,246.721,-61.909,-177.056,6.614,148.347
C02541=1212.002,246.472,-61.882,-177.058,6.611,148.347
C02542=1212.006,246.224,-61.856,-177.060,6.610,148.347
C02543=1212.010,245.975,-61.830,-177.063,6.608,148.347
C02544=1212.015,245.726,-61.803,-177.065,6.606,148.347
C02545=1212.019,245.478,-61.777,-177.068,6.603,148.348
C02546=1212.024,245.229,-61.750,-177.071,6.601,148.348
C02547=1212.028,244.981,-61.724,-177.073,6.599,148.348
C02548=1212.033,244.732,-61.698,-177.076,6.597,148.348
C02549=1212.037,244.484,-61.671,-177.078,6.595,148.349
C02550=1212.041,244.235,-61.646,-177.080,6.593,148.349
C02551=1212.046,243.987,-61.619,-177.084,6.590,148.349
C02552=1212.050,243.738,-61.593,-177.086,6.588,148.349
C02553=1212.055,243.490,-61.566,-177.088,6.586,148.349
C02554=1212.059,243.241,-61.540,-177.091,6.584,148.350
C02555=1212.063,242.992,-61.514,-177.094,6.582,148.350
C02556=1212.068,242.744,-61.487,-177.096,6.580,148.350
C02557=1212.072,242.495,-61.462,-177.098,6.578,148.350
C02558=1212.077,242.247,-61.436,-177.102,6.576,148.351
C02559=1212.082,241.998,-61.409,-177.104,6.574,148.351
C02560=1212.086,241.749,-61.383,-177.106,6.572,148.351
C02561=1212.090,241.500,-61.358,-177.109,6.570,148.351
C02562=1212.095,241.252,-61.331,-177.112,6.568,148.352
C02563=1212.099,241.003,-61.305,-177.114,6.566,148.352
C02564=1212.104,240.755,-61.279,-177.116,6.564,148.352
C02565=1212.109,240.506,-61.253,-177.120,6.561,148.352
C02566=1212.113,240.258,-61.227,-177.122,6.559,148.353
C02567=1212.117,240.009,-61.201,-177.124,6.557,148.353
C02568=1212.121,239.760,-61.175,-177.127,6.555,148.353
C02569=1212.127,239.512,-61.149,-177.129,6.553,148.353
C02570=1212.131,239.264,-61.123,-177.132,6.551,148.354
C02571=1212.135,239.015,-61.097,-177.134,6.549,148.354
C02572=1212.140,238.766,-61.071,-177.137,6.548,148.354
C02573=1212.145,238.518,-61.045,-177.140,6.545,148.354
C02574=1212.149,238.269,-61.019,-177.142,6.543,148.355
C02575=1212.153,238.021,-60.993,-177.145,6.541,148.355
C02576=1212.157,237.772,-60.967,-177.147,6.539,148.355
C02577=1212.163,237.500,-60.939,-177.150,6.537,148.355
C02578=1212.168,237.228,-60.911,-177.153,6.534,148.356
C02579=1212.172,236.957,-60.882,-177.156,6.532,148.356
C02580=1212.178,236.686,-60.854,-177.158,6.530,148.356
C02581=1212.182,236.437,-60.829,-177.161,6.528,148.357
C02582=1212.186,236.188,-60.803,-177.163,6.526,148.357
C02583=1212.191,235.940,-60.778,-177.166,6.524,148.357
C02584=1212.195,235.691,-60.752,-177.169,6.522,148.357
C02585=1212.200,235.442,-60.725,-177.171,6.520,148.358
C02586=1212.204,235.193,-60.700,-177.174,6.518,148.358
C02587=1212.209,234.945,-60.674,-177.176,6.516,148.358
C02588=1212.213,234.697,-60.649,-177.179,6.514,148.358
C02589=1212.218,234.448,-60.623,-177.181,6.512,148.359
C02590=1212.222,234.200,-60.597,-177.184,6.510,148.359
C02591=1212.227,233.951,-60.572,-177.187,6.507,148.359
C02592=1212.231,233.702,-60.546,-177.189,6.506,148.359
C02593=1212.235,233.453,-60.520,-177.192,6.504,148.360
C02594=1212.241,233.205,-60.494,-177.194,6.502,148.360
C02595=1212.245,232.956,-60.468,-177.197,6.500,148.360
C02596=1212.249,232.707,-60.443,-177.199,6.498,148.360
C02597=1212.254,232.459,-60.417,-177.202,6.496,148.361
C02598=1212.258,232.210,-60.392,-177.204,6.494,148.361
C02599=1212.262,231.961,-60.366,-177.207,6.492,148.361
C02600=1212.267,231.713,-60.340,-177.209,6.490,148.362
C02601=1212.271,231.465,-60.315,-177.212,6.488,148.362
C02602=1212.276,231.216,-60.290,-177.215,6.485,148.362
C02603=1212.281,230.967,-60.264,-177.217,6.483,148.362
C02604=1212.285,230.718,-60.239,-177.220,6.482,148.363
C02605=1212.290,230.470,-60.213,-177.223,6.480,148.363
C02606=1212.294,230.221,-60.187,-177.225,6.478,148.363
C02607=1212.299,229.972,-60.162,-177.227,6.476,148.363
C02608=1212.303,229.724,-60.137,-177.230,6.474,148.364
C02609=1212.308,229.475,-60.111,-177.233,6.472,148.364
C02610=1212.312,229.227,-60.086,-177.235,6.470,148.364
C02611=1212.317,228.977,-60.061,-177.237,6.468,148.364
C02612=1212.321,228.729,-60.035,-177.240,6.466,148.365
C02613=1212.326,228.481,-60.010,-177.243,6.464,148.365
C02614=1212.330,228.232,-59.984,-177.245,6.462,148.365
C02615=1212.335,227.983,-59.960,-177.248,6.461,148.366
C02616=1212.339,227.735,-59.934,-177.250,6.458,148.366
C02617=1212.343,227.486,-59.908,-177.253,6.456,148.366
C02618=1212.348,227.237,-59.884,-177.256,6.454,148.366
C02619=1212.352,226.988,-59.858,-177.259,6.452,148.367
C02620=1212.357,226.740,-59.833,-177.261,6.450,148.367
C02621=1212.362,226.491,-59.808,-177.264,6.448,148.367
C02622=1212.367,226.243,-59.782,-177.266,6.446,148.367
C02623=1212.371,225.994,-59.756,-177.269,6.444,148.368
C02624=1212.375,225.745,-59.732,-177.271,6.442,148.368
C02625=1212.379,225.497,-59.707,-177.274,6.441,148.368
C02626=1212.384,225.247,-59.682,-177.277,6.439,148.369
C02627=1212.389,224.999,-59.656,-177.279,6.437,148.369
C02628=1212.393,224.750,-59.631,-177.281,6.435,148.369
C02629=1212.398,224.501,-59.606,-177.284,6.433,148.370
C02630=1212.402,224.253,-59.581,-177.287,6.431,148.370
C02631=1212.407,224.004,-59.556,-177.289,6.429,148.370
C02632=1212.411,223.755,-59.530,-177.292,6.427,148.370
C02633=1212.416,223.507,-59.505,-177.294,6.425,148.371
C02634=1212.420,223.258,-59.480,-177.297,6.423,148.371
C02635=1212.425,223.010,-59.456,-177.299,6.421,148.371
C02636=1212.429,222.761,-59.430,-177.302,6.420,148.372
C02637=1212.434,222.512,-59.405,-177.305,6.418,148.372
C02638=1212.439,222.263,-59.380,-177.308,6.415,148.372
C02639=1212.443,222.015,-59.355,-177.310,6.413,148.372
C02640=1212.447,221.765,-59.330,-177.313,6.411,148.373
C02641=1212.452,221.517,-59.305,-177.315,6.409,148.373
C02642=1212.456,221.268,-59.281,-177.318,6.407,148.373
C02643=1212.461,221.020,-59.255,-177.320,6.406,148.374
C02644=1212.466,220.771,-59.230,-177.323,6.404,148.374
C02645=1212.470,220.522,-59.205,-177.326,6.402,148.374
C02646=1212.474,220.274,-59.181,-177.328,6.400,148.375
C02647=1212.479,220.025,-59.156,-177.331,6.398,148.375
C02648=1212.484,219.776,-59.131,-177.333,6.396,148.375
C02649=1212.488,219.527,-59.106,-177.336,6.394,148.375
C02650=1212.493,219.279,-59.081,-177.338,6.392,148.376
C02651=1212.498,219.030,-59.056,-177.341,6.390,148.376
C02652=1212.501,218.782,-59.031,-177.344,6.389,148.376
C02653=1212.506,218.533,-59.007,-177.346,6.387,148.377
C02654=1212.510,218.284,-58.982,-177.349,6.385,148.377
C02655=1212.515,218.035,-58.958,-177.351,6.383,148.377
C02656=1212.520,217.786,-58.932,-177.354,6.381,148.377
C02657=1212.524,217.538,-58.908,-177.356,6.379,148.378
C02658=1212.529,217.289,-58.883,-177.359,6.377,148.378
C02659=1212.533,217.040,-58.859,-177.362,6.375,148.378
C02660=1212.538,216.791,-58.834,-177.364,6.374,148.379
C02661=1212.543,216.543,-58.809,-177.367,6.372,148.379
C02662=1212.547,216.294,-58.784,-177.370,6.370,148.379
C02663=1212.552,216.045,-58.759,-177.372,6.368,148.380
C02664=1212.556,215.796,-58.735,-177.374,6.366,148.380
C02665=1212.561,215.547,-58.710,-177.377,6.364,148.380
C02666=1212.565,215.299,-58.686,-177.380,6.362,148.381
C02667=1212.569,215.050,-58.660,-177.382,6.360,148.381
C02668=1212.574,214.802,-58.636,-177.385,6.358,148.381
C02669=1212.579,214.553,-58.612,-177.388,6.357,148.382
C02670=1212.583,214.304,-58.587,-177.390,6.355,148.382
C02671=1212.588,214.055,-58.563,-177.393,6.353,148.382
C02672=1212.592,213.807,-58.539,-177.395,6.351,148.383
C02673=1212.597,213.557,-58.514,-177.398,6.349,148.383
C02674=1212.601,213.309,-58.489,-177.401,6.347,148.383
C02675=1212.606,213.060,-58.465,-177.403,6.345,148.383
C02676=1212.610,212.811,-58.440,-177.406,6.343,148.384
C02677=1212.615,212.562,-58.416,-177.408,6.342,148.384
C02678=1212.620,212.314,-58.392,-177.411,6.340,148.384
C02679=1212.625,212.065,-58.367,-177.413,6.338,148.385
C02680=1212.628,211.816,-58.342,-177.416,6.336,148.385
C02681=1212.634,211.546,-58.316,-177.419,6.334,148.385
C02682=1212.639,211.276,-58.289,-177.421,6.332,148.386
C02683=1212.644,211.005,-58.263,-177.425,6.330,148.386
C02684=1212.648,210.734,-58.237,-177.428,6.328,148.387
C02685=1212.653,210.486,-58.212,-177.430,6.326,148.387
C02686=1212.658,210.237,-58.188,-177.433,6.324,148.387
C02687=1212.663,209.989,-58.163,-177.435,6.322,148.387
C02688=1212.667,209.739,-58.139,-177.438,6.320,148.388
C02689=1212.671,209.491,-58.115,-177.440,6.319,148.388
C02690=1212.676,209.242,-58.090,-177.443,6.317,148.388
C02691=1212.681,208.993,-58.067,-177.446,6.315,148.389
C02692=1212.685,208.744,-58.042,-177.448,6.313,148.389
C02693=1212.690,208.495,-58.018,-177.451,6.311,148.389
C02694=1212.694,208.247,-57.993,-177.454,6.309,148.390
C02695=1212.699,207.998,-57.969,-177.456,6.308,148.390
C02696=1212.704,207.750,-57.945,-177.458,6.307,148.390
C02697=1212.708,207.500,-57.921,-177.461,6.305,148.391
C02698=1212.712,207.252,-57.897,-177.464,6.303,148.391
C02699=1212.717,207.003,-57.872,-177.466,6.301,148.391
C02700=1212.722,206.755,-57.848,-177.469,6.299,148.392
C02701=1212.726,206.506,-57.825,-177.472,6.297,148.392
C02702=1212.731,206.256,-57.800,-177.474,6.296,148.392
C02703=1212.735,206.008,-57.776,-177.477,6.294,148.393
C02704=1212.740,205.759,-57.752,-177.480,6.292,148.393
C02705=1212.744,205.510,-57.728,-177.482,6.290,148.393
C02706=1212.749,205.262,-57.704,-177.485,6.288,148.394
C02707=1212.754,205.013,-57.680,-177.487,6.286,148.394
C02708=1212.758,204.763,-57.656,-177.490,6.285,148.394
C02709=1212.762,204.515,-57.632,-177.492,6.282,148.395
C02710=1212.767,204.266,-57.607,-177.495,6.281,148.395
C02711=1212.772,204.017,-57.584,-177.498,6.279,148.395
C02712=1212.777,203.769,-57.560,-177.500,6.277,148.396
C02713=1212.781,203.520,-57.536,-177.502,6.276,148.396
C02714=1212.785,203.271,-57.512,-177.505,6.274,148.396
C02715=1212.789,203.022,-57.488,-177.508,6.272,148.397
C02716=1212.795,202.773,-57.464,-177.510,6.270,148.397
C02717=1212.799,202.525,-57.440,-177.513,6.269,148.397
C02718=1212.804,202.276,-57.416,-177.515,6.267,148.398
C02719=1212.808,202.027,-57.392,-177.518,6.265,148.398
C02720=1212.813,201.779,-57.368,-177.521,6.263,148.398
C02721=1212.817,201.530,-57.345,-177.523,6.261,148.399
C02722=1212.823,201.281,-57.320,-177.526,6.259,148.399
C02723=1212.827,201.031,-57.296,-177.529,6.258,148.399
C02724=1212.831,200.783,-57.272,-177.531,6.256,148.400
C02725=1212.836,200.534,-57.249,-177.533,6.255,148.400
C02726=1212.840,200.285,-57.225,-177.536,6.253,148.400
C02727=1212.845,200.036,-57.202,-177.539,6.251,148.401
C02728=1212.850,199.787,-57.178,-177.541,6.249,148.401
C02729=1212.854,199.539,-57.154,-177.544,6.247,148.401
C02730=1212.859,199.290,-57.131,-177.547,6.246,148.402
C02731=1212.863,199.041,-57.107,-177.549,6.244,148.402
C02732=1212.868,198.792,-57.083,-177.552,6.242,148.403
C02733=1212.872,198.544,-57.059,-177.555,6.240,148.403
C02734=1212.878,198.295,-57.035,-177.557,6.239,148.403
C02735=1212.882,198.046,-57.012,-177.559,6.237,148.404
C02736=1212.887,197.797,-56.988,-177.562,6.235,148.404
C02737=1212.891,197.548,-56.965,-177.565,6.234,148.404
C02738=1212.896,197.299,-56.941,-177.568,6.232,148.405
C02739=1212.901,197.051,-56.917,-177.570,6.230,148.405
C02740=1212.905,196.802,-56.894,-177.573,6.228,148.406
C02741=1212.910,196.553,-56.870,-177.576,6.227,148.406
C02742=1212.914,196.304,-56.846,-177.578,6.225,148.406
C02743=1212.919,196.055,-56.823,-177.580,6.224,148.407
C02744=1212.924,195.806,-56.800,-177.583,6.222,148.407
C02745=1212.928,195.558,-56.776,-177.586,6.220,148.407
C02746=1212.932,195.309,-56.753,-177.588,6.218,148.408
C02747=1212.937,195.060,-56.729,-177.591,6.216,148.408
C02748=1212.941,194.811,-56.706,-177.594,6.215,148.408
C02749=1212.946,194.563,-56.682,-177.596,6.213,148.409
C02750=1212.951,194.314,-56.659,-177.599,6.211,148.409
C02751=1212.955,194.065,-56.635,-177.601,6.210,148.409
C02752=1212.960,193.815,-56.612,-177.604,6.208,148.410
C02753=1212.965,193.566,-56.589,-177.606,6.206,148.410
C02754=1212.969,193.318,-56.564,-177.609,6.204,148.410
C02755=1212.974,193.069,-56.541,-177.612,6.203,148.411
C02756=1212.978,192.820,-56.518,-177.614,6.201,148.411
C02757=1212.983,192.571,-56.494,-177.617,6.199,148.411
C02758=1212.987,192.322,-56.472,-177.619,6.198,148.412
C02759=1212.992,192.073,-56.448,-177.622,6.196,148.412
C02760=1212.997,191.824,-56.425,-177.624,6.194,148.413
C02761=1213.001,191.575,-56.402,-177.627,6.193,148.413
C02762=1213.006,191.327,-56.377,-177.630,6.191,148.413
C02763=1213.010,191.078,-56.354,-177.633,6.189,148.414
C02764=1213.016,190.829,-56.331,-177.635,6.188,148.414
C02765=1213.020,190.581,-56.308,-177.638,6.186,148.415
C02766=1213.024,190.332,-56.285,-177.640,6.184,148.415
C02767=1213.029,190.083,-56.262,-177.643,6.183,148.415
C02768=1213.034,189.834,-56.238,-177.645,6.181,148.416
C02769=1213.038,189.584,-56.215,-177.648,6.179,148.416
C02770=1213.042,189.336,-56.192,-177.650,6.178,148.416
C02771=1213.047,189.087,-56.169,-177.653,6.176,148.417
C02772=1213.052,188.838,-56.145,-177.656,6.174,148.417
C02773=1213.057,188.589,-56.122,-177.658,6.172,148.417
C02774=1213.061,188.341,-56.100,-177.661,6.171,148.418
C02775=1213.066,188.092,-56.076,-177.664,6.169,148.418
C02776=1213.070,187.843,-56.053,-177.666,6.168,148.419
C02777=1213.075,187.594,-56.030,-177.669,6.166,148.419
C02778=1213.079,187.345,-56.007,-177.671,6.165,148.419
C02779=1213.084,187.095,-55.984,-177.674,6.163,148.420
C02780=1213.089,186.847,-55.961,-177.677,6.161,148.420
C02781=1213.094,186.598,-55.938,-177.679,6.160,148.420
C02782=1213.098,186.349,-55.915,-177.681,6.158,148.421
C02783=1213.103,186.100,-55.892,-177.684,6.156,148.421
C02784=1213.107,185.851,-55.868,-177.687,6.154,148.421
C02785=1213.112,185.582,-55.844,-177.690,6.153,148.422
C02786=1213.117,185.312,-55.819,-177.692,6.151,148.422
C02787=1213.123,185.042,-55.794,-177.695,6.149,148.423
C02788=1213.127,184.773,-55.769,-177.698,6.148,148.423
C02789=1213.132,184.524,-55.746,-177.701,6.146,148.424
C02790=1213.136,184.276,-55.724,-177.704,6.144,148.424
C02791=1213.141,184.026,-55.701,-177.706,6.143,148.424
C02792=1213.146,183.777,-55.678,-177.708,6.141,148.425
C02793=1213.150,183.528,-55.655,-177.711,6.139,148.425
C02794=1213.155,183.280,-55.632,-177.714,6.138,148.425
C02795=1213.159,183.031,-55.609,-177.716,6.136,148.426
C02796=1213.164,182.781,-55.586,-177.718,6.135,148.426
C02797=1213.169,182.532,-55.563,-177.722,6.133,148.427
C02798=1213.173,182.284,-55.540,-177.724,6.132,148.427
C02799=1213.179,182.035,-55.518,-177.727,6.130,148.428
C02800=1213.183,181.786,-55.495,-177.730,6.128,148.428
C02801=1213.187,181.537,-55.472,-177.732,6.127,148.428
C02802=1213.192,181.288,-55.450,-177.734,6.125,148.429
C02803=1213.197,181.039,-55.427,-177.737,6.123,148.429
C02804=1213.202,180.790,-55.404,-177.740,6.121,148.429
C02805=1213.206,180.541,-55.382,-177.742,6.121,148.430
C02806=1213.211,180.293,-55.359,-177.745,6.119,148.430
C02807=1213.215,180.044,-55.336,-177.747,6.117,148.431
C02808=1213.220,179.794,-55.313,-177.750,6.115,148.431
C02809=1213.224,179.546,-55.290,-177.753,6.114,148.431
C02810=1213.230,179.297,-55.268,-177.755,6.113,148.432
C02811=1213.234,179.048,-55.245,-177.758,6.111,148.432
C02812=1213.239,178.798,-55.223,-177.761,6.109,148.433
C02813=1213.243,178.550,-55.200,-177.763,6.107,148.433
C02814=1213.248,178.301,-55.177,-177.765,6.106,148.433
C02815=1213.252,178.052,-55.155,-177.768,6.105,148.434
C02816=1213.257,177.804,-55.132,-177.771,6.103,148.434
C02817=1213.262,177.554,-55.110,-177.773,6.101,148.434
C02818=1213.266,177.305,-55.087,-177.775,6.100,148.435
C02819=1213.271,177.056,-55.065,-177.779,6.098,148.435
C02820=1213.275,176.808,-55.042,-177.781,6.097,148.436
C02821=1213.280,176.558,-55.019,-177.784,6.095,148.436
C02822=1213.285,176.309,-54.998,-177.786,6.094,148.437
C02823=1213.289,176.061,-54.975,-177.789,6.092,148.437
C02824=1213.294,175.811,-54.952,-177.791,6.090,148.437
C02825=1213.299,175.563,-54.930,-177.794,6.089,148.438
C02826=1213.304,175.313,-54.907,-177.797,6.088,148.438
C02827=1213.308,175.065,-54.884,-177.799,6.086,148.439
C02828=1213.313,174.816,-54.863,-177.802,6.084,148.439
C02829=1213.318,174.566,-54.840,-177.804,6.083,148.439
C02830=1213.322,174.318,-54.818,-177.807,6.081,148.440
C02831=1213.326,174.069,-54.796,-177.810,6.080,148.440
C02832=1213.331,173.819,-54.773,-177.812,6.078,148.441
C02833=1213.336,173.571,-54.751,-177.815,6.077,148.441
C02834=1213.340,173.322,-54.729,-177.817,6.075,148.441
C02835=1213.346,173.073,-54.706,-177.820,6.073,148.442
C02836=1213.350,172.824,-54.684,-177.823,6.072,148.442
C02837=1213.354,172.575,-54.662,-177.825,6.071,148.443
C02838=1213.360,172.326,-54.639,-177.828,6.069,148.443
C02839=1213.364,172.077,-54.616,-177.830,6.067,148.443
C02840=1213.369,171.829,-54.595,-177.833,6.066,148.444
C02841=1213.374,171.579,-54.572,-177.835,6.064,148.444
C02842=1213.378,171.330,-54.550,-177.838,6.063,148.445
C02843=1213.382,171.082,-54.528,-177.841,6.061,148.445
C02844=1213.387,170.832,-54.506,-177.843,6.060,148.446
C02845=1213.392,170.583,-54.483,-177.846,6.058,148.446
C02846=1213.396,170.334,-54.461,-177.848,6.057,148.446
C02847=1213.401,170.085,-54.440,-177.851,6.056,148.447
C02848=1213.405,169.837,-54.417,-177.854,6.054,148.447
C02849=1213.411,169.588,-54.395,-177.856,6.052,148.448
C02850=1213.415,169.338,-54.373,-177.859,6.050,148.448
C02851=1213.420,169.090,-54.351,-177.861,6.049,148.448
C02852=1213.424,168.840,-54.329,-177.864,6.048,148.449
C02853=1213.430,168.591,-54.307,-177.867,6.046,148.449
C02854=1213.434,168.342,-54.284,-177.869,6.045,148.450
C02855=1213.439,168.094,-54.262,-177.872,6.043,148.450
C02856=1213.443,167.845,-54.240,-177.874,6.042,148.450
C02857=1213.448,167.596,-54.218,-177.877,6.041,148.451
C02858=1213.452,167.347,-54.196,-177.880,6.039,148.451
C02859=1213.458,167.098,-54.174,-177.882,6.037,148.452
C02860=1213.462,166.848,-54.152,-177.884,6.036,148.452
C02861=1213.467,166.600,-54.130,-177.888,6.035,148.453
C02862=1213.471,166.350,-54.108,-177.890,6.033,148.453
C02863=1213.476,166.102,-54.087,-177.892,6.032,148.453
C02864=1213.480,165.852,-54.065,-177.895,6.030,148.454
C02865=1213.485,165.604,-54.043,-177.898,6.028,148.454
C02866=1213.489,165.355,-54.021,-177.900,6.028,148.455
C02867=1213.495,165.106,-53.999,-177.903,6.026,148.455
C02868=1213.499,164.856,-53.976,-177.906,6.024,148.456
C02869=1213.504,164.608,-53.955,-177.908,6.022,148.456
C02870=1213.509,164.359,-53.933,-177.911,6.022,148.457
C02871=1213.513,164.110,-53.911,-177.913,6.020,148.457
C02872=1213.518,163.861,-53.889,-177.916,6.018,148.457
C02873=1213.522,163.612,-53.867,-177.918,6.017,148.458
C02874=1213.527,163.363,-53.846,-177.921,6.016,148.458
C02875=1213.532,163.114,-53.824,-177.923,6.015,148.459
C02876=1213.536,162.865,-53.802,-177.926,6.013,148.459
C02877=1213.541,162.616,-53.780,-177.929,6.011,148.459
C02878=1213.546,162.366,-53.759,-177.931,6.010,148.460
C02879=1213.551,162.118,-53.737,-177.934,6.009,148.460
C02880=1213.555,161.868,-53.715,-177.937,6.007,148.461
C02881=1213.560,161.620,-53.693,-177.939,6.006,148.461
C02882=1213.565,161.371,-53.672,-177.942,6.004,148.462
C02883=1213.569,161.122,-53.650,-177.945,6.002,148.462
C02884=1213.574,160.873,-53.629,-177.947,6.002,148.462
C02885=1213.579,160.623,-53.607,-177.949,6.000,148.463
C02886=1213.583,160.375,-53.585,-177.953,5.998,148.463
C02887=1213.588,160.126,-53.563,-177.955,5.997,148.464
C02888=1213.593,159.877,-53.541,-177.957,5.995,148.464
C02889=1213.598,159.607,-53.518,-177.960,5.994,148.465
C02890=1213.603,159.338,-53.495,-177.963,5.992,148.465
C02891=1213.608,159.069,-53.471,-177.965,5.991,148.466
C02892=1213.613,158.800,-53.448,-177.968,5.990,148.466
C02893=1213.618,158.552,-53.427,-177.971,5.988,148.467
C02894=1213.623,158.302,-53.406,-177.974,5.986,148.467
C02895=1213.627,158.053,-53.384,-177.976,5.985,148.468
C02896=1213.632,157.804,-53.362,-177.979,5.984,148.468
C02897=1213.637,157.555,-53.341,-177.981,5.983,148.468
C02898=1213.641,157.306,-53.319,-177.984,5.981,148.469
C02899=1213.646,157.057,-53.297,-177.987,5.979,148.469
C02900=1213.651,156.808,-53.277,-177.989,5.978,148.470
C02901=1213.655,156.559,-53.255,-177.992,5.977,148.470
C02902=1213.660,156.310,-53.233,-177.995,5.975,148.471
C02903=1213.665,156.061,-53.212,-177.997,5.974,148.471
C02904=1213.670,155.812,-53.191,-178.000,5.972,148.471
C02905=1213.674,155.563,-53.168,-178.002,5.972,148.472
C02906=1213.679,155.314,-53.148,-178.005,5.970,148.472
C02907=1213.683,155.065,-53.126,-178.008,5.968,148.473
C02908=1213.688,154.816,-53.105,-178.010,5.967,148.473
C02909=1213.693,154.567,-53.083,-178.013,5.966,148.474
C02910=1213.698,154.318,-53.062,-178.015,5.965,148.474
C02911=1213.703,154.069,-53.041,-178.018,5.963,148.474
C02912=1213.707,153.819,-53.020,-178.021,5.961,148.475
C02913=1213.712,153.571,-52.998,-178.023,5.960,148.475
C02914=1213.717,153.321,-52.977,-178.025,5.959,148.476
C02915=1213.722,153.073,-52.956,-178.028,5.958,148.476
C02916=1213.725,152.823,-52.935,-178.031,5.956,148.477
C02917=1213.730,152.575,-52.913,-178.033,5.954,148.477
C02918=1213.735,152.325,-52.892,-178.036,5.953,148.478
C02919=1213.740,152.077,-52.871,-178.039,5.952,148.478
C02920=1213.745,151.828,-52.850,-178.041,5.951,148.479
C02921=1213.749,151.578,-52.828,-178.043,5.949,148.479
C02922=1213.754,151.329,-52.807,-178.047,5.948,148.480
C02923=1213.759,151.080,-52.786,-178.049,5.947,148.480
C02924=1213.764,150.831,-52.765,-178.051,5.945,148.480
C02925=1213.768,150.582,-52.744,-178.054,5.944,148.481
C02926=1213.773,150.333,-52.722,-178.057,5.943,148.481
C02927=1213.777,150.084,-52.702,-178.059,5.942,148.482
C02928=1213.782,149.835,-52.680,-178.062,5.940,148.482
C02929=1213.787,149.586,-52.659,-178.065,5.938,148.483
C02930=1213.792,149.337,-52.639,-178.067,5.937,148.483
C02931=1213.796,149.088,-52.617,-178.070,5.936,148.484
C02932=1213.801,148.838,-52.596,-178.072,5.935,148.484
C02933=1213.806,148.590,-52.575,-178.075,5.933,148.484
C02934=1213.811,148.341,-52.554,-178.077,5.932,148.485
C02935=1213.816,148.092,-52.533,-178.080,5.931,148.485
C02936=1213.820,147.843,-52.512,-178.083,5.929,148.486
C02937=1213.825,147.593,-52.491,-178.085,5.928,148.486
C02938=1213.830,147.344,-52.469,-178.088,5.926,148.487
C02939=1213.834,147.095,-52.449,-178.090,5.925,148.487
C02940=1213.839,146.846,-52.428,-178.093,5.924,148.488
C02941=1213.844,146.597,-52.408,-178.095,5.923,148.488
C02942=1213.849,146.348,-52.386,-178.098,5.921,148.489
C02943=1213.854,146.099,-52.365,-178.101,5.921,148.489
C02944=1213.858,145.849,-52.344,-178.103,5.919,148.490
C02945=1213.863,145.600,-52.323,-178.106,5.917,148.490
C02946=1213.867,145.352,-52.302,-178.108,5.916,148.491
C02947=1213.872,145.103,-52.281,-178.111,5.915,148.491
C02948=1213.877,144.854,-52.261,-178.113,5.914,148.491
C02949=1213.882,144.604,-52.240,-178.116,5.912,148.492
C02950=1213.886,144.355,-52.220,-178.119,5.911,148.492
C02951=1213.891,144.106,-52.199,-178.122,5.910,148.493
C02952=1213.896,143.857,-52.178,-178.124,5.909,148.493
C02953=1213.901,143.609,-52.157,-178.126,5.907,148.494
C02954=1213.904,143.359,-52.136,-178.129,5.906,148.494
C02955=1213.910,143.110,-52.115,-178.132,5.905,148.495
C02956=1213.914,142.861,-52.094,-178.134,5.904,148.495
C02957=1213.919,142.611,-52.073,-178.137,5.902,148.496
C02958=1213.924,142.362,-52.053,-178.140,5.900,148.496
C02959=1213.929,142.113,-52.032,-178.142,5.899,148.497
C02960=1213.933,141.864,-52.012,-178.145,5.898,148.497
C02961=1213.938,141.615,-51.991,-178.147,5.897,148.498
C02962=1213.943,141.366,-51.970,-178.150,5.895,148.498
C02963=1213.948,141.117,-51.949,-178.152,5.894,148.499
C02964=1213.953,140.868,-51.929,-178.155,5.893,148.499
C02965=1213.957,140.619,-51.909,-178.158,5.892,148.500
C02966=1213.962,140.370,-51.888,-178.160,5.890,148.500
C02967=1213.967,140.121,-51.867,-178.162,5.889,148.500
C02968=1213.972,139.871,-51.846,-178.166,5.888,148.501
C02969=1213.976,139.622,-51.826,-178.168,5.887,148.501
C02970=1213.981,139.373,-51.805,-178.171,5.885,148.502
C02971=1213.986,139.124,-51.785,-178.173,5.884,148.502
C02972=1213.990,138.875,-51.764,-178.176,5.883,148.503
C02973=1213.995,138.626,-51.743,-178.178,5.882,148.503
C02974=1214.000,138.377,-51.723,-178.181,5.880,148.504
C02975=1214.004,138.128,-51.703,-178.184,5.880,148.504
C02976=1214.009,137.879,-51.682,-178.186,5.878,148.505
C02977=1214.014,137.630,-51.661,-178.188,5.877,148.505
C02978=1214.019,137.380,-51.642,-178.191,5.875,148.506
C02979=1214.024,137.131,-51.621,-178.194,5.874,148.506
C02980=1214.028,136.882,-51.600,-178.197,5.873,148.507
C02981=1214.033,136.633,-51.580,-178.199,5.872,148.507
C02982=1214.038,136.384,-51.559,-178.202,5.870,148.508
C02983=1214.042,136.135,-51.539,-178.204,5.870,148.508
C02984=1214.047,135.886,-51.518,-178.207,5.868,148.509
C02985=1214.052,135.636,-51.498,-178.209,5.867,148.509
C02986=1214.057,135.387,-51.478,-178.212,5.865,148.510
C02987=1214.061,135.138,-51.457,-178.214,5.864,148.510
C02988=1214.066,134.889,-51.436,-178.217,5.863,148.511
C02989=1214.071,134.639,-51.417,-178.219,5.862,148.511
C02990=1214.075,134.390,-51.396,-178.223,5.861,148.512
C02991=1214.080,134.142,-51.376,-178.225,5.860,148.512
C02992=1214.086,133.893,-51.355,-178.228,5.858,148.513
C02993=1214.090,133.624,-51.334,-178.230,5.857,148.513
C02994=1214.095,133.355,-51.311,-178.233,5.856,148.514
C02995=1214.100,133.087,-51.290,-178.236,5.854,148.514
C02996=1214.106,132.818,-51.268,-178.239,5.853,148.515
C02997=1214.110,132.569,-51.248,-178.241,5.852,148.515
C02998=1214.116,132.319,-51.227,-178.244,5.851,148.516
C02999=1214.120,132.071,-51.207,-178.246,5.849,148.516
C03000=1214.125,131.821,-51.187,-178.249,5.848,148.517
C03001=1214.130,131.573,-51.167,-178.252,5.847,148.517
C03002=1214.134,131.324,-51.147,-178.254,5.846,148.518
C03003=1214.139,131.074,-51.127,-178.256,5.845,148.518
C03004=1214.144,130.825,-51.106,-178.259,5.843,148.519
C03005=1214.149,130.576,-51.086,-178.262,5.843,148.519
C03006=1214.153,130.326,-51.066,-178.264,5.841,148.520
C03007=1214.158,130.077,-51.046,-178.267,5.840,148.520
C03008=1214.163,129.829,-51.027,-178.270,5.839,148.521
C03009=1214.167,129.580,-51.006,-178.272,5.838,148.521
C03010=1214.173,129.330,-50.986,-178.275,5.836,148.522
C03011=1214.177,129.081,-50.966,-178.277,5.835,148.522
C03012=1214.182,128.832,-50.945,-178.280,5.834,148.523
C03013=1214.187,128.582,-50.926,-178.282,5.833,148.523
C03014=1214.192,128.334,-50.906,-178.285,5.832,148.524
C03015=1214.196,128.084,-50.886,-178.288,5.830,148.524
C03016=1214.201,127.836,-50.866,-178.290,5.830,148.525
C03017=1214.206,127.586,-50.846,-178.293,5.828,148.525
C03018=1214.210,127.337,-50.825,-178.296,5.827,148.526
C03019=1214.215,127.087,-50.806,-178.298,5.826,148.526
C03020=1214.220,126.839,-50.786,-178.301,5.825,148.527
C03021=1214.225,126.590,-50.766,-178.303,5.824,148.527
C03022=1214.230,126.340,-50.746,-178.306,5.822,148.528
C03023=1214.234,126.091,-50.726,-178.308,5.822,148.528
C03024=1214.240,125.842,-50.706,-178.311,5.820,148.529
C03025=1214.244,125.593,-50.686,-178.314,5.819,148.529
C03026=1214.249,125.343,-50.666,-178.316,5.817,148.530
C03027=1214.253,125.094,-50.646,-178.319,5.817,148.530
C03028=1214.258,124.845,-50.626,-178.321,5.816,148.531
C03029=1214.263,124.596,-50.607,-178.324,5.814,148.531
C03030=1214.268,124.347,-50.587,-178.326,5.813,148.532
C03031=1214.273,124.098,-50.567,-178.329,5.812,148.532
C03032=1214.277,123.848,-50.547,-178.332,5.811,148.533
C03033=1214.282,123.600,-50.527,-178.335,5.810,148.533
C03034=1214.287,123.350,-50.508,-178.337,5.809,148.534
C03035=1214.292,123.101,-50.488,-178.339,5.808,148.534
C03036=1214.296,122.852,-50.468,-178.342,5.806,148.535
C03037=1214.301,122.603,-50.449,-178.345,5.806,148.535
C03038=1214.306,122.353,-50.429,-178.347,5.804,148.536
C03039=1214.310,122.105,-50.409,-178.350,5.803,148.536
C03040=1214.315,121.856,-50.390,-178.352,5.802,148.537
C03041=1214.320,121.606,-50.370,-178.355,5.801,148.537
C03042=1214.325,121.357,-50.350,-178.357,5.800,148.538
C03043=1214.329,121.108,-50.330,-178.360,5.798,148.538
C03044=1214.335,120.859,-50.311,-178.363,5.797,148.539
C03045=1214.339,120.609,-50.291,-178.365,5.797,148.539
C03046=1214.344,120.360,-50.271,-178.368,5.795,148.540
C03047=1214.349,120.111,-50.251,-178.370,5.794,148.540
C03048=1214.353,119.862,-50.232,-178.373,5.793,148.541
C03049=1214.358,119.613,-50.212,-178.375,5.792,148.541
C03050=1214.363,119.364,-50.193,-178.378,5.791,148.542
C03051=1214.368,119.114,-50.174,-178.381,5.789,148.542
C03052=1214.373,118.865,-50.154,-178.383,5.789,148.543
C03053=1214.378,118.616,-50.134,-178.385,5.788,148.543
C03054=1214.383,118.367,-50.114,-178.389,5.786,148.544
C03055=1214.387,118.117,-50.095,-178.391,5.785,148.545
C03056=1214.392,117.869,-50.076,-178.394,5.784,148.545
C03057=1214.397,117.619,-50.056,-178.396,5.783,148.546
C03058=1214.401,117.369,-50.037,-178.399,5.782,148.546
C03059=1214.407,117.121,-50.017,-178.402,5.781,148.547
C03060=1214.412,116.871,-49.998,-178.404,5.780,148.547
C03061=1214.416,116.622,-49.979,-178.407,5.779,148.548
C03062=1214.421,116.374,-49.959,-178.409,5.778,148.548
C03063=1214.425,116.124,-49.939,-178.412,5.777,148.549
C03064=1214.431,115.875,-49.920,-178.415,5.775,148.549
C03065=1214.435,115.626,-49.901,-178.417,5.775,148.550
C03066=1214.439,115.376,-49.881,-178.419,5.774,148.550
C03067=1214.445,115.127,-49.862,-178.423,5.772,148.551
C03068=1214.450,114.878,-49.842,-178.425,5.771,148.551
C03069=1214.455,114.629,-49.823,-178.427,5.771,148.552
C03070=1214.459,114.380,-49.804,-178.430,5.769,148.552
C03071=1214.464,114.131,-49.784,-178.433,5.768,148.553
C03072=1214.469,113.881,-49.765,-178.435,5.767,148.553
C03073=1214.473,113.632,-49.746,-178.438,5.766,148.554
C03074=1214.478,113.383,-49.726,-178.440,5.765,148.555
C03075=1214.483,113.134,-49.707,-178.443,5.764,148.555
C03076=1214.489,112.884,-49.688,-178.445,5.763,148.556
C03077=1214.493,112.635,-49.669,-178.448,5.762,148.556
C03078=1214.498,112.386,-49.650,-178.451,5.760,148.557
C03079=1214.503,112.136,-49.630,-178.453,5.760,148.557
C03080=1214.507,111.887,-49.611,-178.456,5.759,148.558
C03081=1214.512,111.638,-49.592,-178.458,5.757,148.558
C03082=1214.517,111.389,-49.572,-178.461,5.757,148.559
C03083=1214.521,111.140,-49.553,-178.463,5.756,148.559
C03084=1214.526,110.891,-49.534,-178.466,5.754,148.560
C03085=1214.532,110.641,-49.515,-178.469,5.753,148.560
C03086=1214.536,110.392,-49.496,-178.471,5.753,148.561
C03087=1214.541,110.143,-49.477,-178.474,5.751,148.561
C03088=1214.545,109.894,-49.458,-178.476,5.750,148.562
C03089=1214.551,109.645,-49.438,-178.479,5.749,148.562
C03090=1214.555,109.395,-49.419,-178.482,5.748,148.563
C03091=1214.560,109.146,-49.401,-178.484,5.747,148.564
C03092=1214.565,108.896,-49.381,-178.486,5.746,148.564
C03093=1214.570,108.648,-49.362,-178.490,5.745,148.565
C03094=1214.574,108.398,-49.343,-178.492,5.744,148.565
C03095=1214.580,108.149,-49.324,-178.494,5.743,148.566
C03096=1214.584,107.900,-49.305,-178.497,5.742,148.566
C03097=1214.589,107.632,-49.284,-178.500,5.741,148.567
C03098=1214.595,107.362,-49.264,-178.503,5.740,148.568
C03099=1214.599,107.095,-49.244,-178.506,5.739,148.568
C03100=1214.604,106.826,-49.223,-178.508,5.737,148.569
C03101=1214.610,106.577,-49.204,-178.511,5.737,148.569
C03102=1214.614,106.327,-49.185,-178.513,5.736,148.570
C03103=1214.619,106.079,-49.166,-178.516,5.735,148.570
C03104=1214.624,105.829,-49.148,-178.519,5.734,148.571
C03105=1214.629,105.580,-49.128,-178.521,5.733,148.571
C03106=1214.634,105.331,-49.110,-178.523,5.732,148.572
C03107=1214.639,105.081,-49.091,-178.526,5.730,148.572
C03108=1214.643,104.832,-49.072,-178.529,5.730,148.573
C03109=1214.648,104.583,-49.052,-178.531,5.729,148.574
C03110=1214.653,104.334,-49.034,-178.534,5.727,148.574
C03111=1214.658,104.085,-49.015,-178.537,5.727,148.575
C03112=1214.663,103.835,-48.997,-178.539,5.726,148.575
C03113=1214.668,103.586,-48.977,-178.542,5.724,148.576
C03114=1214.672,103.337,-48.958,-178.544,5.723,148.576
C03115=1214.678,103.087,-48.940,-178.547,5.723,148.577
C03116=1214.682,102.839,-48.921,-178.549,5.722,148.577
C03117=1214.687,102.589,-48.903,-178.552,5.720,148.578
C03118=1214.692,102.340,-48.883,-178.555,5.720,148.579
C03119=1214.696,102.090,-48.865,-178.557,5.719,148.579
C03120=1214.702,101.841,-48.846,-178.560,5.718,148.580
C03121=1214.706,101.592,-48.828,-178.563,5.717,148.580
C03122=1214.711,101.343,-48.808,-178.565,5.716,148.581
C03123=1214.716,101.093,-48.790,-178.567,5.715,148.581
C03124=1214.720,100.844,-48.771,-178.570,5.714,148.582
C03125=1214.726,100.595,-48.753,-178.573,5.713,148.582
C03126=1214.730,100.346,-48.734,-178.575,5.712,148.583
C03127=1214.735,100.096,-48.715,-178.578,5.711,148.583
C03128=1214.740,99.847,-48.696,-178.581,5.710,148.584
C03129=1214.745,99.598,-48.678,-178.583,5.709,148.584
C03130=1214.749,99.349,-48.659,-178.585,5.709,148.585
C03131=1214.755,99.099,-48.641,-178.589,5.707,148.586
C03132=1214.760,98.850,-48.623,-178.591,5.706,148.586
C03133=1214.764,98.601,-48.603,-178.593,5.706,148.587
C03134=1214.769,98.352,-48.585,-178.595,5.705,148.587
C03135=1214.774,98.103,-48.566,-178.599,5.703,148.588
C03136=1214.778,97.853,-48.548,-178.601,5.703,148.589
C03137=1214.784,97.604,-48.529,-178.603,5.702,148.589
C03138=1214.788,97.355,-48.511,-178.606,5.701,148.590
C03139=1214.793,97.105,-48.492,-178.609,5.699,148.590
C03140=1214.798,96.856,-48.474,-178.611,5.699,148.591
C03141=1214.803,96.607,-48.455,-178.614,5.698,148.591
C03142=1214.808,96.358,-48.437,-178.616,5.697,148.592
C03143=1214.812,96.108,-48.419,-178.619,5.696,148.592
C03144=1214.817,95.859,-48.399,-178.622,5.695,148.593
C03145=1214.822,95.610,-48.381,-178.624,5.694,148.593
C03146=1214.827,95.360,-48.363,-178.627,5.694,148.594
C03147=1214.832,95.111,-48.345,-178.629,5.692,148.594
C03148=1214.837,94.862,-48.326,-178.632,5.691,148.595
C03149=1214.842,94.613,-48.308,-178.635,5.691,148.596
C03150=1214.846,94.363,-48.289,-178.637,5.690,148.596
C03151=1214.851,94.114,-48.272,-178.640,5.688,148.597
C03152=1214.856,93.865,-48.252,-178.642,5.688,148.597
C03153=1214.861,93.616,-48.234,-178.645,5.687,148.598
C03154=1214.866,93.366,-48.216,-178.647,5.686,148.599
C03155=1214.871,93.117,-48.198,-178.650,5.684,148.599
C03156=1214.875,92.868,-48.180,-178.653,5.684,148.600
C03157=1214.881,92.619,-48.161,-178.655,5.683,148.600
C03158=1214.885,92.369,-48.142,-178.657,5.682,148.601
C03159=1214.890,92.120,-48.124,-178.660,5.681,148.601
C03160=1214.895,91.871,-48.106,-178.663,5.680,148.602
C03161=1214.900,91.621,-48.088,-178.665,5.679,148.602
C03162=1214.904,91.371,-48.070,-178.668,5.679,148.603
C03163=1214.910,91.123,-48.051,-178.670,5.678,148.604
C03164=1214.914,90.873,-48.033,-178.673,5.676,148.604
C03165=1214.919,90.624,-48.015,-178.676,5.676,148.605
C03166=1214.924,90.375,-47.997,-178.678,5.675,148.605
C03167=1214.929,90.125,-47.978,-178.681,5.674,148.606
C03168=1214.933,89.876,-47.960,-178.684,5.673,148.606
C03169=1214.938,89.627,-47.942,-178.686,5.672,148.607
C03170=1214.943,89.378,-47.925,-178.688,5.671,148.608
C03171=1214.948,89.129,-47.907,-178.691,5.671,148.608
C03172=1214.954,88.879,-47.888,-178.693,5.670,148.609
C03173=1214.958,88.629,-47.870,-178.696,5.669,148.609
C03174=1214.963,88.380,-47.852,-178.699,5.668,148.610
C03175=1214.968,88.131,-47.834,-178.701,5.667,148.610
C03176=1214.973,87.882,-47.816,-178.704,5.666,148.611
C03177=1214.978,87.632,-47.798,-178.707,5.665,148.612
C03178=1214.983,87.383,-47.780,-178.709,5.664,148.612
C03179=1214.987,87.133,-47.761,-178.712,5.663,148.613
C03180=1214.992,86.884,-47.743,-178.714,5.663,148.613
C03181=1214.997,86.635,-47.725,-178.717,5.662,148.614
C03182=1215.002,86.386,-47.707,-178.720,5.661,148.614
C03183=1215.007,86.137,-47.689,-178.722,5.660,148.615
C03184=1215.012,85.888,-47.671,-178.724,5.659,148.616
C03185=1215.017,85.638,-47.653,-178.727,5.658,148.616
C03186=1215.021,85.389,-47.635,-178.730,5.658,148.617
C03187=1215.026,85.139,-47.617,-178.732,5.657,148.617
C03188=1215.031,84.890,-47.599,-178.735,5.656,148.618
C03189=1215.036,84.641,-47.581,-178.738,5.655,148.619
C03190=1215.040,84.392,-47.563,-178.740,5.654,148.619
C03191=1215.045,84.143,-47.545,-178.742,5.653,148.620
C03192=1215.051,83.893,-47.528,-178.745,5.653,148.620
C03193=1215.056,83.644,-47.510,-178.748,5.651,148.621
C03194=1215.060,83.394,-47.492,-178.750,5.651,148.621
C03195=1215.065,83.145,-47.474,-178.753,5.650,148.622
C03196=1215.070,82.896,-47.456,-178.755,5.649,148.622
C03197=1215.075,82.647,-47.438,-178.758,5.648,148.623
C03198=1215.080,82.396,-47.420,-178.761,5.647,148.624
C03199=1215.084,82.148,-47.403,-178.763,5.646,148.624
C03200=1215.089,81.898,-47.385,-178.766,5.646,148.625
C03201=1215.094,81.630,-47.366,-178.768,5.645,148.625
C03202=1215.100,81.362,-47.347,-178.772,5.644,148.626
C03203=1215.105,81.094,-47.328,-178.774,5.643,148.627
C03204=1215.110,80.825,-47.309,-178.777,5.642,148.627
C03205=1215.115,80.576,-47.291,-178.779,5.641,148.628
C03206=1215.120,80.326,-47.273,-178.782,5.640,148.628
C03207=1215.125,80.077,-47.255,-178.785,5.639,148.629
C03208=1215.130,79.828,-47.237,-178.787,5.639,148.630
C03209=1215.135,79.578,-47.220,-178.789,5.638,148.630
C03210=1215.140,79.329,-47.202,-178.792,5.637,148.631
C03211=1215.144,79.080,-47.185,-178.795,5.637,148.632
C03212=1215.150,78.830,-47.167,-178.797,5.635,148.632
C03213=1215.154,78.581,-47.149,-178.800,5.634,148.633
C03214=1215.159,78.332,-47.131,-178.803,5.634,148.633
C03215=1215.165,78.082,-47.114,-178.805,5.633,148.634
C03216=1215.170,77.833,-47.096,-178.807,5.632,148.634
C03217=1215.174,77.584,-47.079,-178.810,5.632,148.635
C03218=1215.179,77.335,-47.062,-178.812,5.631,148.635
C03219=1215.184,77.085,-47.044,-178.815,5.629,148.636
C03220=1215.189,76.836,-47.026,-178.818,5.629,148.637
C03221=1215.193,76.587,-47.009,-178.821,5.628,148.637
C03222=1215.198,76.337,-46.991,-178.823,5.627,148.638
C03223=1215.203,76.088,-46.974,-178.825,5.627,148.639
C03224=1215.208,75.839,-46.956,-178.828,5.626,148.639
C03225=1215.213,75.589,-46.938,-178.830,5.625,148.640
C03226=1215.218,75.340,-46.921,-178.833,5.624,148.640
C03227=1215.223,75.091,-46.903,-178.836,5.623,148.641
C03228=1215.228,74.841,-46.886,-178.839,5.623,148.642
C03229=1215.232,74.592,-46.868,-178.841,5.622,148.642
C03230=1215.237,74.342,-46.851,-178.843,5.621,148.643
C03231=1215.242,74.093,-46.833,-178.846,5.621,148.643
C03232=1215.247,73.843,-46.816,-178.848,5.620,148.644
C03233=1215.251,73.594,-46.799,-178.851,5.618,148.644
C03234=1215.257,73.345,-46.781,-178.854,5.618,148.645
C03235=1215.262,73.095,-46.763,-178.857,5.617,148.646
C03236=1215.266,72.846,-46.747,-178.859,5.616,148.646
C03237=1215.272,72.597,-46.729,-178.861,5.616,148.647
C03238=1215.277,72.348,-46.712,-178.864,5.615,148.647
C03239=1215.281,72.099,-46.694,-178.866,5.614,148.648
C03240=1215.286,71.849,-46.677,-178.869,5.614,148.649
C03241=1215.291,71.599,-46.660,-178.872,5.612,148.649
C03242=1215.296,71.350,-46.642,-178.875,5.612,148.650
C03243=1215.301,71.101,-46.625,-178.877,5.611,148.650
C03244=1215.306,70.851,-46.607,-178.879,5.610,148.651
C03245=1215.310,70.602,-46.591,-178.882,5.610,148.652
C03246=1215.316,70.353,-46.574,-178.885,5.609,148.652
C03247=1215.321,70.104,-46.556,-178.887,5.608,148.653
C03248=1215.325,69.854,-46.539,-178.889,5.608,148.653
C03249=1215.330,69.605,-46.521,-178.892,5.607,148.654
C03250=1215.335,69.355,-46.504,-178.895,5.606,148.655
C03251=1215.340,69.106,-46.487,-178.897,5.605,148.655
C03252=1215.345,68.857,-46.469,-178.900,5.604,148.656
C03253=1215.349,68.607,-46.452,-178.903,5.604,148.656
C03254=1215.355,68.358,-46.436,-178.905,5.603,148.657
C03255=1215.359,68.109,-46.418,-178.907,5.602,148.658
C03256=1215.365,67.859,-46.401,-178.910,5.601,148.658
C03257=1215.369,67.610,-46.384,-178.913,5.601,148.659
C03258=1215.374,67.360,-46.367,-178.915,5.600,148.659
C03259=1215.379,67.111,-46.350,-178.917,5.599,148.660
C03260=1215.384,66.862,-46.333,-178.921,5.598,148.661
C03261=1215.390,66.612,-46.315,-178.923,5.597,148.661
C03262=1215.394,66.363,-46.299,-178.925,5.597,148.662
C03263=1215.399,66.114,-46.281,-178.928,5.596,148.662
C03264=1215.403,65.864,-46.264,-178.931,5.595,148.663
C03265=1215.409,65.615,-46.247,-178.933,5.595,148.664
C03266=1215.414,65.366,-46.231,-178.935,5.594,148.664
C03267=1215.419,65.116,-46.213,-178.938,5.593,148.665
C03268=1215.423,64.867,-46.196,-178.941,5.593,148.665
C03269=1215.428,64.617,-46.179,-178.943,5.592,148.666
C03270=1215.433,64.368,-46.162,-178.946,5.591,148.667
C03271=1215.439,64.118,-46.145,-178.949,5.590,148.667
C03272=1215.443,63.869,-46.128,-178.951,5.589,148.668
C03273=1215.447,63.620,-46.111,-178.954,5.589,148.669
C03274=1215.453,63.371,-46.094,-178.957,5.588,148.669
C03275=1215.458,63.122,-46.077,-178.959,5.587,148.670
C03276=1215.463,62.872,-46.060,-178.961,5.587,148.670
C03277=1215.467,62.622,-46.043,-178.964,5.586,148.671
C03278=1215.473,62.372,-46.026,-178.967,5.586,148.672
C03279=1215.478,62.124,-46.010,-178.969,5.585,148.672
C03280=1215.483,61.874,-45.993,-178.971,5.584,148.673
C03281=1215.487,61.624,-45.976,-178.974,5.584,148.673
C03282=1215.492,61.376,-45.960,-178.977,5.583,148.674
C03283=1215.497,61.126,-45.942,-178.979,5.582,148.674
C03284=1215.502,60.877,-45.925,-178.981,5.582,148.675
C03285=1215.507,60.627,-45.908,-178.985,5.580,148.676
C03286=1215.512,60.378,-45.891,-178.987,5.580,148.676
C03287=1215.517,60.129,-45.875,-178.990,5.579,148.677
C03288=1215.522,59.879,-45.858,-178.992,5.578,148.678
C03289=1215.526,59.630,-45.841,-178.995,5.578,148.678
C03290=1215.531,59.381,-45.825,-178.997,5.577,148.679
C03291=1215.537,59.131,-45.807,-179.000,5.576,148.680
C03292=1215.541,58.882,-45.791,-179.002,5.575,148.680
C03293=1215.546,58.633,-45.774,-179.005,5.575,148.681
C03294=1215.551,58.383,-45.757,-179.007,5.574,148.681
C03295=1215.556,58.134,-45.740,-179.010,5.574,148.682
C03296=1215.561,57.885,-45.724,-179.013,5.573,148.683
C03297=1215.566,57.635,-45.707,-179.015,5.572,148.683
C03298=1215.571,57.385,-45.691,-179.017,5.572,148.684
C03299=1215.576,57.136,-45.675,-179.020,5.571,148.684
C03300=1215.581,56.886,-45.657,-179.023,5.571,148.685
C03301=1215.586,56.637,-45.641,-179.025,5.570,148.686
C03302=1215.591,56.388,-45.624,-179.027,5.569,148.686
C03303=1215.596,56.138,-45.607,-179.030,5.569,148.687
C03304=1215.600,55.889,-45.590,-179.033,5.568,148.688
C03305=1215.606,55.621,-45.573,-179.036,5.567,148.688
C03306=1215.611,55.351,-45.555,-179.039,5.566,148.689
C03307=1215.617,55.083,-45.537,-179.041,5.566,148.690
C03308=1215.622,54.816,-45.519,-179.044,5.565,148.690
C03309=1215.627,54.566,-45.503,-179.047,5.564,148.691
C03310=1215.632,54.316,-45.486,-179.049,5.564,148.691
C03311=1215.637,54.067,-45.470,-179.051,5.563,148.692
C03312=1215.641,53.817,-45.453,-179.054,5.562,148.693
C03313=1215.646,53.568,-45.436,-179.057,5.562,148.693
C03314=1215.652,53.318,-45.420,-179.059,5.561,148.694
C03315=1215.657,53.069,-45.403,-179.061,5.560,148.694
C03316=1215.662,52.820,-45.387,-179.064,5.560,148.695
C03317=1215.666,52.571,-45.371,-179.067,5.558,148.696
C03318=1215.671,52.321,-45.354,-179.070,5.558,148.696
C03319=1215.677,52.071,-45.338,-179.072,5.557,148.697
C03320=1215.681,51.822,-45.321,-179.075,5.556,148.698
C03321=1215.686,51.573,-45.305,-179.077,5.556,148.698
C03322=1215.691,51.324,-45.288,-179.080,5.555,148.699
C03323=1215.696,51.074,-45.272,-179.083,5.555,148.700
C03324=1215.701,50.825,-45.256,-179.085,5.554,148.700
C03325=1215.705,50.575,-45.239,-179.087,5.553,148.701
C03326=1215.711,50.325,-45.223,-179.090,5.553,148.701
C03327=1215.716,50.076,-45.206,-179.093,5.552,148.702
C03328=1215.721,49.827,-45.190,-179.095,5.552,148.703
C03329=1215.726,49.577,-45.174,-179.098,5.551,148.703
C03330=1215.731,49.328,-45.158,-179.100,5.550,148.704
C03331=1215.735,49.079,-45.141,-179.103,5.550,148.704
C03332=1215.740,48.829,-45.125,-179.105,5.549,148.705
C03333=1215.745,48.580,-45.109,-179.108,5.549,148.706
C03334=1215.750,48.330,-45.092,-179.111,5.548,148.706
C03335=1215.756,48.081,-45.076,-179.113,5.547,148.707
C03336=1215.760,47.831,-45.059,-179.115,5.547,148.708
C03337=1215.765,47.582,-45.044,-179.118,5.546,148.708
C03338=1215.770,47.332,-45.027,-179.121,5.545,148.709
C03339=1215.775,47.084,-45.011,-179.123,5.545,148.710
C03340=1215.780,46.834,-44.995,-179.126,5.544,148.710
C03341=1215.785,46.585,-44.978,-179.128,5.543,148.711
C03342=1215.790,46.335,-44.962,-179.131,5.543,148.711
C03343=1215.795,46.086,-44.946,-179.133,5.542,148.712
C03344=1215.800,45.836,-44.930,-179.136,5.542,148.713
C03345=1215.805,45.587,-44.914,-179.139,5.541,148.713
C03346=1215.809,45.337,-44.898,-179.141,5.541,148.714
C03347=1215.814,45.088,-44.882,-179.143,5.540,148.714
C03348=1215.819,44.838,-44.866,-179.146,5.539,148.715
C03349=1215.824,44.589,-44.849,-179.149,5.539,148.716
C03350=1215.829,44.339,-44.833,-179.151,5.538,148.716
C03351=1215.834,44.090,-44.817,-179.154,5.538,148.717
C03352=1215.839,43.840,-44.801,-179.157,5.537,148.718
C03353=1215.844,43.591,-44.785,-179.159,5.536,148.718
C03354=1215.849,43.342,-44.769,-179.161,5.536,148.719
C03355=1215.854,43.093,-44.753,-179.163,5.536,148.720
C03356=1215.859,42.843,-44.737,-179.166,5.535,148.720
C03357=1215.864,42.594,-44.720,-179.169,5.535,148.721
C03358=1215.869,42.344,-44.705,-179.171,5.534,148.722
C03359=1215.874,42.094,-44.689,-179.173,5.533,148.722
C03360=1215.879,41.845,-44.673,-179.176,5.533,148.723
C03361=1215.884,41.595,-44.657,-179.179,5.532,148.723
C03362=1215.889,41.346,-44.640,-179.181,5.532,148.724
C03363=1215.894,41.097,-44.625,-179.184,5.531,148.725
C03364=1215.899,40.847,-44.609,-179.187,5.531,148.725
C03365=1215.904,40.598,-44.592,-179.189,5.530,148.726
C03366=1215.908,40.348,-44.577,-179.191,5.529,148.727
C03367=1215.914,40.099,-44.561,-179.194,5.529,148.727
C03368=1215.919,39.850,-44.545,-179.197,5.528,148.728
C03369=1215.924,39.600,-44.529,-179.199,5.527,148.729
C03370=1215.929,39.351,-44.514,-179.202,5.527,148.729
C03371=1215.933,39.101,-44.497,-179.204,5.526,148.730
C03372=1215.939,38.852,-44.481,-179.207,5.525,148.730
C03373=1215.944,38.602,-44.466,-179.209,5.525,148.731
C03374=1215.949,38.353,-44.449,-179.212,5.524,148.732
C03375=1215.953,38.104,-44.434,-179.215,5.524,148.732
C03376=1215.959,37.854,-44.419,-179.217,5.523,148.733
C03377=1215.963,37.604,-44.403,-179.220,5.523,148.734
C03378=1215.969,37.356,-44.386,-179.222,5.522,148.734
C03379=1215.973,37.105,-44.370,-179.225,5.521,148.735
C03380=1215.979,36.856,-44.355,-179.227,5.521,148.736
C03381=1215.983,36.607,-44.340,-179.230,5.521,148.736
C03382=1215.988,36.357,-44.323,-179.232,5.520,148.737
C03383=1215.993,36.108,-44.307,-179.235,5.520,148.738
C03384=1215.999,35.859,-44.292,-179.237,5.519,148.738
C03385=1216.003,35.609,-44.276,-179.240,5.518,148.739
C03386=1216.008,35.359,-44.261,-179.242,5.518,148.739
C03387=1216.013,35.111,-44.245,-179.245,5.517,148.740
C03388=1216.018,34.861,-44.229,-179.248,5.517,148.741
C03389=1216.023,34.611,-44.213,-179.250,5.516,148.741
C03390=1216.029,34.362,-44.198,-179.253,5.516,148.742
C03391=1216.033,34.112,-44.182,-179.255,5.515,148.743
C03392=1216.038,33.863,-44.167,-179.258,5.514,148.743
C03393=1216.043,33.613,-44.151,-179.260,5.514,148.744
C03394=1216.048,33.364,-44.134,-179.263,5.513,148.745
C03395=1216.053,33.115,-44.119,-179.266,5.513,148.745
C03396=1216.058,32.865,-44.104,-179.268,5.512,148.746
C03397=1216.063,32.616,-44.088,-179.270,5.512,148.747
C03398=1216.068,32.366,-44.072,-179.272,5.512,148.747
C03399=1216.073,32.117,-44.057,-179.275,5.511,148.748
C03400=1216.078,31.867,-44.042,-179.278,5.510,148.748
C03401=1216.083,31.617,-44.026,-179.280,5.510,148.749
C03402=1216.088,31.368,-44.011,-179.283,5.509,148.750
C03403=1216.093,31.119,-43.995,-179.286,5.509,148.750
C03404=1216.098,30.869,-43.979,-179.288,5.508,148.751
C03405=1216.102,30.619,-43.964,-179.291,5.508,148.752
C03406=1216.108,30.370,-43.949,-179.293,5.507,148.752
C03407=1216.113,30.121,-43.933,-179.296,5.506,148.753
C03408=1216.118,29.872,-43.918,-179.298,5.506,148.754
C03409=1216.123,29.602,-43.901,-179.301,5.505,148.754
C03410=1216.128,29.334,-43.884,-179.304,5.505,148.755
C03411=1216.134,29.065,-43.867,-179.306,5.504,148.756
C03412=1216.139,28.797,-43.851,-179.309,5.504,148.757
C03413=1216.144,28.547,-43.835,-179.312,5.503,148.757
C03414=1216.149,28.298,-43.820,-179.314,5.503,148.758
C03415=1216.154,28.048,-43.804,-179.317,5.502,148.758
C03416=1216.159,27.799,-43.789,-179.319,5.502,148.759
C03417=1216.164,27.549,-43.774,-179.322,5.502,148.760
C03418=1216.169,27.300,-43.758,-179.324,5.501,148.760
C03419=1216.175,27.051,-43.743,-179.327,5.501,148.761
C03420=1216.179,26.801,-43.727,-179.330,5.500,148.762
C03421=1216.184,26.551,-43.712,-179.332,5.499,148.762
C03422=1216.189,26.302,-43.697,-179.334,5.499,148.763
C03423=1216.195,26.052,-43.682,-179.337,5.498,148.764
C03424=1216.199,25.803,-43.667,-179.340,5.498,148.764
C03425=1216.204,25.553,-43.651,-179.342,5.497,148.765
C03426=1216.209,25.304,-43.635,-179.344,5.497,148.766
C03427=1216.214,25.055,-43.620,-179.347,5.497,148.766
C03428=1216.219,24.805,-43.605,-179.350,5.496,148.767
C03429=1216.224,24.556,-43.590,-179.352,5.495,148.767
C03430=1216.230,24.306,-43.575,-179.354,5.495,148.768
C03431=1216.234,24.056,-43.559,-179.357,5.494,148.769
C03432=1216.239,23.807,-43.544,-179.360,5.494,148.769
C03433=1216.244,23.558,-43.529,-179.362,5.493,148.770
C03434=1216.249,23.308,-43.514,-179.365,5.493,148.771
C03435=1216.254,23.059,-43.499,-179.367,5.493,148.771
C03436=1216.260,22.809,-43.483,-179.370,5.493,148.772
C03437=1216.264,22.560,-43.468,-179.372,5.492,148.773
C03438=1216.269,22.310,-43.452,-179.374,5.491,148.773
C03439=1216.274,22.060,-43.438,-179.377,5.491,148.774
C03440=1216.279,21.811,-43.423,-179.380,5.490,148.775
C03441=1216.284,21.562,-43.408,-179.382,5.490,148.775
C03442=1216.290,21.312,-43.393,-179.385,5.489,148.776
C03443=1216.294,21.063,-43.378,-179.387,5.489,148.777
C03444=1216.300,20.813,-43.362,-179.390,5.489,148.777
C03445=1216.304,20.564,-43.347,-179.392,5.488,148.778
C03446=1216.309,20.314,-43.332,-179.395,5.488,148.779
C03447=1216.314,20.065,-43.317,-179.397,5.487,148.779
C03448=1216.319,19.815,-43.302,-179.400,5.486,148.780
C03449=1216.324,19.565,-43.287,-179.403,5.486,148.781
C03450=1216.329,19.316,-43.272,-179.405,5.485,148.781
C03451=1216.334,19.067,-43.256,-179.407,5.486,148.782
C03452=1216.339,18.817,-43.242,-179.410,5.485,148.783
C03453=1216.344,18.568,-43.227,-179.413,5.484,148.783
C03454=1216.349,18.319,-43.212,-179.415,5.484,148.784
C03455=1216.354,18.069,-43.197,-179.418,5.483,148.785
C03456=1216.360,17.820,-43.182,-179.421,5.483,148.785
C03457=1216.364,17.569,-43.167,-179.423,5.482,148.786
C03458=1216.369,17.320,-43.152,-179.425,5.481,148.786
C03459=1216.374,17.071,-43.136,-179.427,5.482,148.787
C03460=1216.379,16.821,-43.122,-179.430,5.481,148.788
C03461=1216.384,16.572,-43.107,-179.433,5.481,148.789
C03462=1216.389,16.322,-43.092,-179.435,5.480,148.789
C03463=1216.394,16.073,-43.077,-179.438,5.480,148.790
C03464=1216.399,15.823,-43.063,-179.441,5.479,148.791
C03465=1216.404,15.574,-43.047,-179.443,5.479,148.791
C03466=1216.409,15.324,-43.033,-179.445,5.479,148.792
C03467=1216.414,15.075,-43.018,-179.447,5.478,148.792
C03468=1216.420,14.825,-43.003,-179.450,5.477,148.793
C03469=1216.424,14.576,-42.988,-179.453,5.477,148.794
C03470=1216.429,14.326,-42.974,-179.455,5.476,148.794
C03471=1216.435,14.077,-42.958,-179.458,5.476,148.795
C03472=1216.440,13.827,-42.944,-179.460,5.476,148.796
C03473=1216.444,13.578,-42.929,-179.463,5.476,148.796
C03474=1216.450,13.328,-42.914,-179.465,5.475,148.797
C03475=1216.455,13.079,-42.899,-179.468,5.475,148.798
C03476=1216.460,12.829,-42.885,-179.471,5.474,148.799
C03477=1216.464,12.580,-42.870,-179.473,5.474,148.799
C03478=1216.470,12.330,-42.855,-179.475,5.474,148.800
C03479=1216.475,12.081,-42.840,-179.478,5.473,148.800
C03480=1216.480,11.831,-42.826,-179.480,5.472,148.801
C03481=1216.485,11.581,-42.812,-179.483,5.472,148.802
C03482=1216.490,11.332,-42.796,-179.486,5.471,148.802
C03483=1216.495,11.082,-42.782,-179.488,5.471,148.803
C03484=1216.500,10.833,-42.767,-179.490,5.471,148.804
C03485=1216.504,10.583,-42.753,-179.493,5.471,148.804
C03486=1216.510,10.333,-42.738,-179.496,5.470,148.805
C03487=1216.515,10.084,-42.723,-179.498,5.470,148.806
C03488=1216.520,9.835,-42.708,-179.501,5.469,148.807
C03489=1216.525,9.585,-42.694,-179.503,5.468,148.807
C03490=1216.529,9.336,-42.679,-179.505,5.469,148.808
C03491=1216.535,9.086,-42.664,-179.508,5.468,148.808
C03492=1216.540,8.836,-42.650,-179.510,5.468,148.809
C03493=1216.545,8.588,-42.635,-179.513,5.467,148.810
C03494=1216.550,8.338,-42.621,-179.516,5.466,148.810
C03495=1216.555,8.088,-42.607,-179.518,5.466,148.811
C03496=1216.560,7.839,-42.592,-179.520,5.466,148.812
C03497=1216.566,7.589,-42.577,-179.523,5.466,148.812
C03498=1216.570,7.339,-42.563,-179.526,5.465,148.813
C03499=1216.575,7.090,-42.548,-179.528,5.465,148.814
C03500=1216.580,6.841,-42.533,-179.531,5.464,148.815
C03501=1216.585,6.591,-42.519,-179.533,5.464,148.815
C03502=1216.590,6.341,-42.505,-179.535,5.464,148.816
C03503=1216.595,6.092,-42.490,-179.538,5.463,148.816
C03504=1216.600,5.842,-42.475,-179.541,5.463,148.817
C03505=1216.606,5.593,-42.461,-179.543,5.462,148.818
C03506=1216.611,5.343,-42.447,-179.546,5.462,148.818
C03507=1216.616,5.094,-42.432,-179.548,5.462,148.819
C03508=1216.620,4.845,-42.418,-179.551,5.461,148.820
C03509=1216.625,4.595,-42.403,-179.553,5.461,148.820
C03510=1216.630,4.345,-42.389,-179.556,5.460,148.821
C03511=1216.635,4.096,-42.375,-179.559,5.460,148.822
C03512=1216.640,3.846,-42.360,-179.561,5.460,148.823
C03513=1216.646,3.578,-42.345,-179.563,5.460,148.823
C03514=1216.652,3.309,-42.329,-179.566,5.459,148.824
C03515=1216.657,3.039,-42.314,-179.569,5.459,148.825
C03516=1216.662,2.770,-42.298,-179.571,5.458,148.825
C03517=1216.667,2.521,-42.284,-179.574,5.457,148.826
C03518=1216.672,2.271,-42.269,-179.577,5.457,148.827
C03519=1216.677,2.021,-42.255,-179.579,5.456,148.827
C03520=1216.683,1.772,-42.241,-179.581,5.457,148.828
C03521=1216.688,1.523,-42.227,-179.584,5.456,148.829
C03522=1216.693,1.273,-42.213,-179.587,5.456,148.829
C03523=1216.698,1.023,-42.198,-179.589,5.455,148.830
C03524=1216.702,0.774,-42.183,-179.592,5.455,148.831
C03525=1216.708,0.525,-42.170,-179.594,5.455,148.831
C03526=1216.713,0.275,-42.155,-179.597,5.454,148.832
C03527=1216.718,0.026,-42.141,-179.599,5.454,148.833
C03528=1216.723,-0.224,-42.127,-179.601,5.453,148.833
C03529=1216.728,-0.474,-42.112,-179.604,5.453,148.834
C03530=1216.733,-0.723,-42.099,-179.606,5.453,148.835
C03531=1216.738,-0.973,-42.084,-179.609,5.452,148.835
C03532=1216.743,-1.222,-42.070,-179.612,5.452,148.836
C03533=1216.748,-1.472,-42.056,-179.614,5.451,148.837
C03534=1216.753,-1.722,-42.041,-179.616,5.452,148.837
C03535=1216.759,-1.971,-42.028,-179.619,5.451,148.838
C03536=1216.764,-2.220,-42.013,-179.622,5.451,148.839
C03537=1216.769,-2.470,-41.999,-179.624,5.450,148.840
C03538=1216.773,-2.719,-41.985,-179.626,5.450,148.840
C03539=1216.778,-2.968,-41.971,-179.629,5.450,148.841
C03540=1216.783,-3.218,-41.957,-179.632,5.449,148.842
C03541=1216.788,-3.468,-41.943,-179.634,5.449,148.842
C03542=1216.794,-3.718,-41.929,-179.636,5.448,148.843
C03543=1216.798,-3.968,-41.915,-179.638,5.448,148.843
C03544=1216.804,-4.217,-41.901,-179.641,5.448,148.844
C03545=1216.809,-4.467,-41.887,-179.644,5.447,148.845
C03546=1216.814,-4.716,-41.873,-179.646,5.447,148.846
C03547=1216.819,-4.965,-41.859,-179.649,5.447,148.846
C03548=1216.824,-5.215,-41.845,-179.651,5.447,148.847
C03549=1216.829,-5.465,-41.831,-179.654,5.446,148.848
C03550=1216.834,-5.714,-41.816,-179.656,5.446,148.848
C03551=1216.839,-5.964,-41.803,-179.659,5.445,148.849
C03552=1216.844,-6.214,-41.789,-179.661,5.445,148.850
C03553=1216.849,-6.463,-41.775,-179.664,5.445,148.850
C03554=1216.854,-6.713,-41.760,-179.667,5.444,148.851
C03555=1216.859,-6.962,-41.747,-179.669,5.444,148.852
C03556=1216.864,-7.211,-41.733,-179.671,5.444,148.852
C03557=1216.869,-7.462,-41.719,-179.674,5.444,148.853
C03558=1216.875,-7.711,-41.705,-179.676,5.443,148.854
C03559=1216.880,-7.960,-41.691,-179.679,5.442,148.854
C03560=1216.884,-8.210,-41.677,-179.681,5.443,148.855
C03561=1216.890,-8.459,-41.663,-179.683,5.442,148.856
C03562=1216.895,-8.709,-41.650,-179.686,5.442,148.856
C03563=1216.900,-8.959,-41.636,-179.689,5.441,148.857
C03564=1216.905,-9.208,-41.622,-179.691,5.441,148.858
C03565=1216.910,-9.457,-41.608,-179.694,5.441,148.858
C03566=1216.915,-9.708,-41.594,-179.696,5.440,148.859
C03567=1216.920,-9.957,-41.581,-179.699,5.440,148.860
C03568=1216.925,-10.206,-41.566,-179.701,5.440,148.860
C03569=1216.930,-10.456,-41.553,-179.704,5.440,148.861
C03570=1216.936,-10.705,-41.539,-179.706,5.439,148.862
C03571=1216.940,-10.955,-41.525,-179.709,5.439,148.863
C03572=1216.945,-11.205,-41.511,-179.711,5.439,148.863
C03573=1216.951,-11.454,-41.498,-179.714,5.438,148.864
C03574=1216.955,-11.704,-41.484,-179.716,5.438,148.865
C03575=1216.960,-11.954,-41.470,-179.719,5.437,148.865
C03576=1216.966,-12.203,-41.457,-179.720,5.437,148.866
C03577=1216.971,-12.453,-41.443,-179.723,5.437,148.866
C03578=1216.975,-12.702,-41.428,-179.726,5.436,148.867
C03579=1216.981,-12.952,-41.415,-179.728,5.436,148.868
C03580=1216.986,-13.201,-41.402,-179.731,5.436,148.869
C03581=1216.991,-13.450,-41.388,-179.733,5.436,148.869
C03582=1216.996,-13.701,-41.374,-179.736,5.435,148.870
C03583=1217.001,-13.950,-41.360,-179.739,5.435,148.871
C03584=1217.006,-14.200,-41.347,-179.741,5.435,148.871
C03585=1217.011,-14.449,-41.333,-179.743,5.435,148.872
C03586=1217.016,-14.698,-41.320,-179.746,5.434,148.873
C03587=1217.021,-14.948,-41.306,-179.748,5.434,148.873
C03588=1217.026,-15.198,-41.292,-179.751,5.434,148.874
C03589=1217.032,-15.447,-41.279,-179.753,5.433,148.875
C03590=1217.037,-15.697,-41.265,-179.756,5.433,148.876
C03591=1217.042,-15.947,-41.252,-179.758,5.433,148.876
C03592=1217.047,-16.196,-41.238,-179.761,5.433,148.877
C03593=1217.052,-16.445,-41.224,-179.763,5.432,148.878
C03594=1217.057,-16.695,-41.211,-179.766,5.432,148.878
C03595=1217.062,-16.945,-41.197,-179.768,5.432,148.879
C03596=1217.067,-17.195,-41.184,-179.770,5.431,148.879
C03597=1217.072,-17.444,-41.170,-179.773,5.431,148.880
C03598=1217.078,-17.694,-41.157,-179.775,5.431,148.881
C03599=1217.082,-17.943,-41.143,-179.778,5.430,148.882
C03600=1217.088,-18.193,-41.130,-179.780,5.430,148.882
C03601=1217.093,-18.442,-41.116,-179.783,5.429,148.883
C03602=1217.098,-18.692,-41.103,-179.785,5.430,148.884
C03603=1217.103,-18.942,-41.090,-179.788,5.429,148.884
C03604=1217.108,-19.191,-41.076,-179.790,5.429,148.885
C03605=1217.113,-19.441,-41.063,-179.792,5.429,148.886
C03606=1217.118,-19.690,-41.049,-179.795,5.429,148.886
C03607=1217.123,-19.940,-41.036,-179.798,5.428,148.887
C03608=1217.128,-20.190,-41.021,-179.800,5.428,148.888
C03609=1217.133,-20.439,-41.009,-179.802,5.428,148.888
C03610=1217.138,-20.689,-40.995,-179.805,5.427,148.889
C03611=1217.143,-20.938,-40.982,-179.808,5.427,148.890
C03612=1217.149,-21.188,-40.968,-179.810,5.427,148.891
C03613=1217.153,-21.437,-40.955,-179.813,5.427,148.891
C03614=1217.159,-21.687,-40.942,-179.815,5.426,148.892
C03615=1217.164,-21.937,-40.929,-179.818,5.426,148.893
C03616=1217.169,-22.186,-40.915,-179.819,5.426,148.893
C03617=1217.174,-22.455,-40.901,-179.823,5.426,148.894
C03618=1217.180,-22.725,-40.886,-179.825,5.425,148.895
C03619=1217.185,-22.995,-40.872,-179.828,5.425,148.895
C03620=1217.191,-23.263,-40.858,-179.831,5.424,148.896
C03621=1217.196,-23.514,-40.845,-179.833,5.424,148.897
C03622=1217.201,-23.763,-40.832,-179.835,5.424,148.898
C03623=1217.206,-24.013,-40.818,-179.838,5.423,148.898
C03624=1217.211,-24.262,-40.805,-179.840,5.424,148.899
C03625=1217.217,-24.512,-40.791,-179.843,5.423,148.900
C03626=1217.221,-24.761,-40.778,-179.845,5.423,148.900
C03627=1217.227,-25.011,-40.765,-179.847,5.423,148.901
C03628=1217.232,-25.261,-40.752,-179.850,5.423,148.902
C03629=1217.237,-25.510,-40.739,-179.853,5.422,148.902
C03630=1217.242,-25.760,-40.725,-179.855,5.422,148.903
C03631=1217.247,-26.009,-40.713,-179.858,5.422,148.904
C03632=1217.252,-26.259,-40.699,-179.860,5.421,148.904
C03633=1217.257,-26.509,-40.686,-179.863,5.421,148.905
C03634=1217.262,-26.758,-40.673,-179.865,5.421,148.906
C03635=1217.267,-27.008,-40.659,-179.868,5.421,148.907
C03636=1217.273,-27.257,-40.647,-179.870,5.420,148.907
C03637=1217.278,-27.507,-40.633,-179.872,5.420,148.908
C03638=1217.283,-27.757,-40.621,-179.875,5.420,148.908
C03639=1217.287,-28.006,-40.607,-179.877,5.419,148.909
C03640=1217.293,-28.256,-40.594,-179.879,5.420,148.910
C03641=1217.297,-28.506,-40.581,-179.882,5.419,148.911
C03642=1217.303,-28.755,-40.568,-179.885,5.419,148.911
C03643=1217.308,-29.005,-40.555,-179.887,5.418,148.912
C03644=1217.313,-29.255,-40.542,-179.889,5.418,148.913
